SPLINE
SPL {X  -158.456, Y  +360.399, Z    +0.000, E1   -16.490, E3 -394778.901}
SPL {X  -159.553, Y  +370.677, Z    +0.000, E1   -10.576, E3 -394786.661}
SPL {X  -159.960, Y  +379.402, Z    +0.000, E1    -5.303, E3 -394790.682}
SPL {X  -159.990, Y  +385.983, Z    +0.000, E1    -0.882, E3 -394792.754}
SPL {X  -159.990, Y  +390.933, Z    +0.000, E1    +2.877, E3 -394794.202}
SPL {X  -159.990, Y  +396.375, Z    +0.000, E1    +7.538, E3 -394795.977}
SPL {X  -159.990, Y  +405.219, Z    +0.000, E1   +15.296, E3 -394800.294}
SPL {X  -159.990, Y  +427.416, Z    +0.000, E1   +29.294, E3 -394821.349}
SPL {X  -159.990, Y  +450.630, Z    +0.000, E1   +34.875, E3 -394862.921}
SPL {X  -159.990, Y  +456.402, Z    +0.000, E1   +35.061, E3 -394879.197}
SPL {X  -159.990, Y  +460.708, Z    +0.000, E1   +35.045, E3 -394892.255}
SPL {X  -159.990, Y  +464.162, Z    +0.000, E1   +35.038, E3 -394902.711}
SPL {X  -159.990, Y  +467.857, Z    +0.000, E1   +35.053, E3 -394913.868}
SPL {X  -159.990, Y  +471.326, Z    +0.000, E1   +35.038, E3 -394924.363}
SPL {X  -159.990, Y  +474.610, Z    +0.000, E1   +35.053, E3 -394934.262}
SPL {X  -159.990, Y  +478.303, Z    +0.000, E1   +35.049, E3 -394945.435}
SPL {X  -159.990, Y  +482.537, Z    +0.000, E1   +35.066, E3 -394958.226}
SPL {X  -159.990, Y  +487.181, Z    +0.000, E1   +35.054, E3 -394972.309}
SPL {X  -159.990, Y  +492.368, Z    +0.000, E1   +35.076, E3 -394987.981}
SPL {X  -159.990, Y  +497.072, Z    +0.000, E1   +35.040, E3 -395002.277}
SPL {X  -159.990, Y  +500.395, Z    +0.000, E1   +35.033, E3 -395012.340}
SPL {X  -159.990, Y  +505.138, Z    +0.000, E1   +35.092, E3 -395026.576}
SPL {X  -159.990, Y  +510.443, Z    +0.000, E1   +35.051, E3 -395042.695}
SPL {X  -159.990, Y  +514.632, Z    +0.000, E1   +35.050, E3 -395055.365}
SPL {X  -159.990, Y  +518.055, Z    +0.000, E1   +35.037, E3 -395065.734}
SPL {X  -159.990, Y  +521.637, Z    +0.000, E1   +35.056, E3 -395076.544}
SPL {X  -159.990, Y  +526.246, Z    +0.000, E1   +35.065, E3 -395090.447}
SPL {X  -159.990, Y  +531.319, Z    +0.000, E1   +35.072, E3 -395105.803}
SPL {X  -159.990, Y  +537.053, Z    +0.000, E1   +35.083, E3 -395123.136}
SPL {X  -159.990, Y  +542.114, Z    +0.000, E1   +35.053, E3 -395138.482}
SPL {X  -159.990, Y  +545.724, Z    +0.000, E1   +35.043, E3 -395149.407}
SPL {X  -159.990, Y  +549.546, Z    +0.000, E1   +35.061, E3 -395160.931}
SPL {X  -159.990, Y  +554.793, Z    +0.000, E1   +35.100, E3 -395176.695}
SPL {X  -159.990, Y  +560.931, Z    +0.000, E1   +35.098, E3 -395195.256}
SPL {X  -159.990, Y  +566.542, Z    +0.000, E1   +35.080, E3 -395212.264}
SPL {X  -159.990, Y  +571.374, Z    +0.000, E1   +35.070, E3 -395226.888}
SPL {X  -159.990, Y  +575.771, Z    +0.000, E1   +35.064, E3 -395240.193}
SPL {X  -159.990, Y  +579.185, Z    +0.000, E1   +35.047, E3 -395250.541}
SPL {X  -159.990, Y  +581.944, Z    +0.000, E1   +35.051, E3 -395258.879}
SPL {X  -159.990, Y  +585.414, Z    +0.000, E1   +35.059, E3 -395269.362}
SPL {X  -159.990, Y  +590.166, Z    +0.000, E1   +35.084, E3 -395283.690}
SPL {X  -159.990, Y  +595.313, Z    +0.000, E1   +35.073, E3 -395299.269}
SPL {X  -159.990, Y  +600.543, Z    +0.000, E1   +35.091, E3 -395315.051}
SPL {X  -159.990, Y  +605.846, Z    +0.000, E1   +35.077, E3 -395331.102}
SPL {X  -159.990, Y  +609.372, Z    +0.000, E1   +35.047, E3 -395341.800}
SPL {X  -159.990, Y  +613.036, Z    +0.000, E1   +35.082, E3 -395352.835}
SPL {X  -159.990, Y  +617.577, Z    +0.000, E1   +35.061, E3 -395366.596}
SPL {X  -159.990, Y  +621.534, Z    +0.000, E1   +35.068, E3 -395378.531}
SPL {X  -159.990, Y  +625.237, Z    +0.000, E1   +35.062, E3 -395389.733}
SPL {X  -159.990, Y  +629.217, Z    +0.000, E1   +35.065, E3 -395401.790}
SPL {X  -159.990, Y  +632.566, Z    +0.000, E1   +35.044, E3 -395411.953}
SPL {X  -159.990, Y  +635.965, Z    +0.000, E1   +35.065, E3 -395422.196}
SPL {X  -159.990, Y  +640.633, Z    +0.000, E1   +35.080, E3 -395436.285}
SPL {X  -159.990, Y  +646.430, Z    +0.000, E1   +35.102, E3 -395453.786}
SPL {X  -159.990, Y  +651.502, Z    +0.000, E1   +35.058, E3 -395469.196}
SPL {X  -159.990, Y  +654.793, Z    +0.000, E1   +35.049, E3 -395479.159}
SPL {X  -159.990, Y  +657.535, Z    +0.000, E1   +35.049, E3 -395487.456}
SPL {X  -159.990, Y  +661.105, Z    +0.000, E1   +35.059, E3 -395498.236}
SPL {X  -159.990, Y  +665.311, Z    +0.000, E1   +35.064, E3 -395510.951}
SPL {X  -159.990, Y  +670.193, Z    +0.000, E1   +35.076, E3 -395525.698}
SPL {X  -159.948, Y  +675.148, Z    +0.000, E1   +35.069, E3 -395540.690}
SPL {X  -159.752, Y  +680.228, Z    +0.000, E1   +35.050, E3 -395556.238}
SPL {X  -159.371, Y  +685.563, Z    +0.000, E1   +34.989, E3 -395572.749}
SPL {X  -158.886, Y  +690.264, Z    +0.000, E1   +34.888, E3 -395587.500}
SPL {X  -158.362, Y  +694.266, Z    +0.000, E1   +34.794, E3 -395600.174}
SPL {X  -157.614, Y  +698.973, Z    +0.000, E1   +34.690, E3 -395615.174}
SPL {X  -156.640, Y  +704.066, Z    +0.000, E1   +34.516, E3 -395631.600}
SPL {X  -155.835, Y  +707.723, Z    +0.000, E1   +34.344, E3 -395643.542}
SPL {X  -155.080, Y  +710.833, Z    +0.000, E1   +34.231, E3 -395653.692}
SPL {X  -153.755, Y  +715.731, Z    +0.000, E1   +30.246, E3 -395702.958}
ENDSPLINE

SPLINE
SPL {X  -155.537, Y  +708.983, Z    +0.000, E1   +25.008, E3 -395728.784}
SPL {X  -158.838, Y  +690.666, Z    +0.000, E1   +14.584, E3 -395753.497}
SPL {X  -159.750, Y  +680.262, Z    +0.000, E1    +8.563, E3 -395759.637}
SPL {X  -159.973, Y  +673.798, Z    +0.000, E1    +4.600, E3 -395762.101}
SPL {X  -159.990, Y  +668.863, Z    +0.000, E1    +1.298, E3 -395763.541}
SPL {X  -159.990, Y  +663.839, Z    +0.000, E1    -2.454, E3 -395764.802}
SPL {X  -159.990, Y  +657.071, Z    +0.000, E1    -8.297, E3 -395766.994}
SPL {X  -159.990, Y  +646.193, Z    +0.000, E1   -17.980, E3 -395772.721}
SPL {X  -159.990, Y  +621.124, Z    +0.000, E1   -32.598, E3 -395796.208}
SPL {X  -159.990, Y  +597.855, Z    +0.000, E1   -36.862, E3 -395839.127}
SPL {X  -159.990, Y  +592.884, Z    +0.000, E1   -36.865, E3 -395853.198}
SPL {X  -159.990, Y  +587.104, Z    +0.000, E1   -36.878, E3 -395869.555}
SPL {X  -159.990, Y  +581.795, Z    +0.000, E1   -36.847, E3 -395884.654}
SPL {X  -159.990, Y  +576.165, Z    +0.000, E1   -36.887, E3 -395900.533}
SPL {X  -159.990, Y  +570.328, Z    +0.000, E1   -36.855, E3 -395917.106}
SPL {X  -159.990, Y  +566.126, Z    +0.000, E1   -36.841, E3 -395929.012}
SPL {X  -159.990, Y  +562.387, Z    +0.000, E1   -36.853, E3 -395939.545}
SPL {X  -159.990, Y  +557.944, Z    +0.000, E1   -36.859, E3 -395952.139}
SPL {X  -159.990, Y  +553.661, Z    +0.000, E1   -36.844, E3 -395964.303}
SPL {X  -159.990, Y  +549.195, Z    +0.000, E1   -36.856, E3 -395976.938}
SPL {X  -159.990, Y  +543.458, Z    +0.000, E1   -36.882, E3 -395993.136}
SPL {X  -159.990, Y  +538.694, Z    +0.000, E1   -36.835, E3 -396006.720}
SPL {X  -159.990, Y  +534.469, Z    +0.000, E1   -36.855, E3 -396018.666}
SPL {X  -159.990, Y  +530.428, Z    +0.000, E1   -36.821, E3 -396030.199}
SPL {X  -159.990, Y  +525.940, Z    +0.000, E1   -36.859, E3 -396042.846}
SPL {X  -159.990, Y  +520.301, Z    +0.000, E1   -36.855, E3 -396058.822}
SPL {X  -159.990, Y  +516.005, Z    +0.000, E1   -36.824, E3 -396071.048}
SPL {X  -159.990, Y  +512.789, Z    +0.000, E1   -36.824, E3 -396080.156}
SPL {X  -159.990, Y  +508.591, Z    +0.000, E1   -36.846, E3 -396092.019}
SPL {X  -159.990, Y  +503.454, Z    +0.000, E1   -36.847, E3 -396106.574}
SPL {X  -159.990, Y  +498.817, Z    +0.000, E1   -36.830, E3 -396119.757}
SPL {X  -159.990, Y  +498.054, Z    +0.000, E1   -35.692, E3 -396128.871}
ENDSPLINE

SPLINE
SPL {X  -159.990, Y  +505.140, Z    +0.000, E1   -30.523, E3 -396139.898}
ENDSPLINE

SPLINE
SPL {X  -159.990, Y  +497.800, Z    +0.000, E1   -31.845, E3 -396156.854}
SPL {X  -159.990, Y  +492.180, Z    +0.000, E1   -32.851, E3 -396168.990}
SPL {X  -159.990, Y  +486.073, Z    +0.000, E1   -33.960, E3 -396181.625}
SPL {X  -159.990, Y  +477.314, Z    +0.000, E1   -35.342, E3 -396199.803}
SPL {X  -159.990, Y  +471.459, Z    +0.000, E1   -35.779, E3 -396214.343}
SPL {X  -159.990, Y  +467.485, Z    +0.000, E1   -35.768, E3 -396226.072}
SPL {X  -159.990, Y  +462.739, Z    +0.000, E1   -35.799, E3 -396240.000}
SPL {X  -159.990, Y  +457.385, Z    +0.000, E1   -35.788, E3 -396255.784}
SPL {X  -159.990, Y  +452.637, Z    +0.000, E1   -35.783, E3 -396269.776}
SPL {X  -159.990, Y  +446.982, Z    +0.000, E1   -35.815, E3 -396286.377}
SPL {X  -159.990, Y  +442.593, Z    +0.000, E1   -35.759, E3 -396299.386}
SPL {X  -159.990, Y  +439.109, Z    +0.000, E1   -35.781, E3 -396309.603}
SPL {X  -159.990, Y  +435.535, Z    +0.000, E1   -35.764, E3 -396320.154}
SPL {X  -159.990, Y  +431.100, Z    +0.000, E1   -35.807, E3 -396333.139}
SPL {X  -159.990, Y  +426.641, Z    +0.000, E1   -35.769, E3 -396346.326}
SPL {X  -159.990, Y  +422.627, Z    +0.000, E1   -35.788, E3 -396358.123}
SPL {X  -159.990, Y  +417.866, Z    +0.000, E1   -35.788, E3 -396372.137}
SPL {X  -159.990, Y  +413.498, Z    +0.000, E1   -35.779, E3 -396385.019}
SPL {X  -159.990, Y  +408.600, Z    +0.000, E1   -35.802, E3 -396399.406}
SPL {X  -159.990, Y  +403.496, Z    +0.000, E1   -35.787, E3 -396414.461}
SPL {X  -159.990, Y  +398.606, Z    +0.000, E1   -35.794, E3 -396428.848}
SPL {X  -159.990, Y  +394.138, Z    +0.000, E1   -35.778, E3 -396442.032}
SPL {X  -159.990, Y  +388.813, Z    +0.000, E1   -35.819, E3 -396457.644}
SPL {X  -159.990, Y  +383.172, Z    +0.000, E1   -35.789, E3 -396474.298}
SPL {X  -159.936, Y  +378.352, Z    +0.000, E1   -35.782, E3 -396488.537}
SPL {X  -159.790, Y  +374.497, Z    +0.000, E1   -35.735, E3 -396500.081}
SPL {X  -159.547, Y  +370.604, Z    +0.000, E1   -35.724, E3 -396511.766}
SPL {X  -159.134, Y  +365.969, Z    +0.000, E1   -35.644, E3 -396525.852}
SPL {X  -158.606, Y  +361.498, Z    +0.000, E1   -35.550, E3 -396539.616}
SPL {X  -157.918, Y  +356.833, Z    +0.000, E1   -35.439, E3 -396554.069}
SPL {X  -157.185, Y  +352.671, Z    +0.000, E1   -35.292, E3 -396567.129}
SPL {X  -156.302, Y  +348.345, Z    +0.000, E1   -35.165, E3 -396580.750}
SPL {X  -155.054, Y  +343.066, Z    +0.000, E1   -34.964, E3 -396597.565}
SPL {X  -154.305, Y  +340.232, Z    +0.000, E1   -28.975, E3 -396655.125}
ENDSPLINE

SPLINE
SPL {X  -158.456, Y  +360.399, Z    +0.000, E1   -16.490, E3 -396691.945}
SPL {X  -159.553, Y  +370.677, Z    +0.000, E1   -10.576, E3 -396699.705}
SPL {X  -159.960, Y  +379.402, Z    +0.000, E1    -5.303, E3 -396703.725}
SPL {X  -159.990, Y  +387.301, Z    +0.000, E1    -0.001, E3 -396706.186}
SPL {X  -159.990, Y  +392.161, Z    +0.000, E1    +3.946, E3 -396707.598}
SPL {X  -159.990, Y  +396.375, Z    +0.000, E1    +7.538, E3 -396709.020}
SPL {X  -159.990, Y  +404.277, Z    +0.000, E1   +14.543, E3 -396712.683}
SPL {X  -159.990, Y  +423.101, Z    +0.000, E1   +27.351, E3 -396729.122}
SPL {X  -159.990, Y  +430.933, Z    +0.000, E1   +30.672, E3 -396739.093}
SPL {X  -159.990, Y  +451.842, Z    +0.000, E1   +35.050, E3 -396778.464}
SPL {X  -159.990, Y  +456.402, Z    +0.000, E1   +35.061, E3 -396792.240}
SPL {X  -159.990, Y  +460.708, Z    +0.000, E1   +35.045, E3 -396805.298}
SPL {X  -159.990, Y  +464.162, Z    +0.000, E1   +35.038, E3 -396815.754}
SPL {X  -159.990, Y  +467.857, Z    +0.000, E1   +35.053, E3 -396826.911}
SPL {X  -159.990, Y  +471.326, Z    +0.000, E1   +35.038, E3 -396837.406}
SPL {X  -159.990, Y  +474.610, Z    +0.000, E1   +35.053, E3 -396847.306}
SPL {X  -159.990, Y  +478.303, Z    +0.000, E1   +35.049, E3 -396858.478}
SPL {X  -159.990, Y  +482.537, Z    +0.000, E1   +35.066, E3 -396871.269}
SPL {X  -159.990, Y  +487.181, Z    +0.000, E1   +35.054, E3 -396885.352}
SPL {X  -159.990, Y  +490.807, Z    +0.000, E1   +35.036, E3 -396896.354}
SPL {X  -159.990, Y  +493.669, Z    +0.000, E1   +35.034, E3 -396905.033}
SPL {X  -159.990, Y  +497.072, Z    +0.000, E1   +35.040, E3 -396915.320}
SPL {X  -159.990, Y  +501.645, Z    +0.000, E1   +35.067, E3 -396929.103}
SPL {X  -159.990, Y  +507.359, Z    +0.000, E1   +35.080, E3 -396946.360}
SPL {X  -159.990, Y  +512.562, Z    +0.000, E1   +35.055, E3 -396962.142}
SPL {X  -159.990, Y  +517.156, Z    +0.000, E1   +35.059, E3 -396976.024}
SPL {X  -159.990, Y  +521.637, Z    +0.000, E1   +35.056, E3 -396989.587}
SPL {X  -159.990, Y  +525.227, Z    +0.000, E1   +35.041, E3 -397000.448}
SPL {X  -159.990, Y  +529.413, Z    +0.000, E1   +35.072, E3 -397013.077}
SPL {X  -159.990, Y  +534.797, Z    +0.000, E1   +35.069, E3 -397029.377}
SPL {X  -159.990, Y  +538.710, Z    +0.000, E1   +35.033, E3 -397041.274}
SPL {X  -159.990, Y  +542.114, Z    +0.000, E1   +35.053, E3 -397051.526}
SPL {X  -159.990, Y  +546.612, Z    +0.000, E1   +35.065, E3 -397065.097}
SPL {X  -159.990, Y  +551.596, Z    +0.000, E1   +35.079, E3 -397080.132}
SPL {X  -159.990, Y  +557.043, Z    +0.000, E1   +35.087, E3 -397096.554}
SPL {X  -159.990, Y  +562.842, Z    +0.000, E1   +35.098, E3 -397114.087}
SPL {X  -159.990, Y  +568.750, Z    +0.000, E1   +35.087, E3 -397131.972}
SPL {X  -159.990, Y  +574.780, Z    +0.000, E1   +35.101, E3 -397150.183}
SPL {X  -159.990, Y  +580.750, Z    +0.000, E1   +35.087, E3 -397168.259}
SPL {X  -159.990, Y  +585.414, Z    +0.000, E1   +35.059, E3 -397182.405}
SPL {X  -159.990, Y  +588.716, Z    +0.000, E1   +35.047, E3 -397192.408}
SPL {X  -159.990, Y  +592.923, Z    +0.000, E1   +35.084, E3 -397205.072}
SPL {X  -159.990, Y  +598.554, Z    +0.000, E1   +35.088, E3 -397222.091}
SPL {X  -159.990, Y  +603.289, Z    +0.000, E1   +35.068, E3 -397236.419}
SPL {X  -159.990, Y  +607.919, Z    +0.000, E1   +35.079, E3 -397250.408}
SPL {X  -159.990, Y  +613.036, Z    +0.000, E1   +35.082, E3 -397265.878}
SPL {X  -159.990, Y  +617.577, Z    +0.000, E1   +35.061, E3 -397279.640}
SPL {X  -159.990, Y  +621.534, Z    +0.000, E1   +35.068, E3 -397291.574}
SPL {X  -159.990, Y  +626.426, Z    +0.000, E1   +35.093, E3 -397306.333}
SPL {X  -159.990, Y  +631.553, Z    +0.000, E1   +35.068, E3 -397321.891}
SPL {X  -159.990, Y  +636.917, Z    +0.000, E1   +35.095, E3 -397338.070}
SPL {X  -159.990, Y  +641.534, Z    +0.000, E1   +35.053, E3 -397352.098}
SPL {X  -159.990, Y  +646.430, Z    +0.000, E1   +35.102, E3 -397366.829}
SPL {X  -159.990, Y  +651.502, Z    +0.000, E1   +35.058, E3 -397382.239}
SPL {X  -159.990, Y  +654.793, Z    +0.000, E1   +35.049, E3 -397392.203}
SPL {X  -159.990, Y  +657.535, Z    +0.000, E1   +35.049, E3 -397400.499}
SPL {X  -159.990, Y  +661.105, Z    +0.000, E1   +35.059, E3 -397411.279}
SPL {X  -159.990, Y  +665.311, Z    +0.000, E1   +35.064, E3 -397423.994}
SPL {X  -159.990, Y  +670.193, Z    +0.000, E1   +35.076, E3 -397438.741}
SPL {X  -159.948, Y  +675.148, Z    +0.000, E1   +35.069, E3 -397453.733}
SPL {X  -159.752, Y  +680.228, Z    +0.000, E1   +35.050, E3 -397469.281}
SPL {X  -159.371, Y  +685.563, Z    +0.000, E1   +34.989, E3 -397485.793}
SPL {X  -158.886, Y  +690.264, Z    +0.000, E1   +34.888, E3 -397500.544}
SPL {X  -158.362, Y  +694.266, Z    +0.000, E1   +34.794, E3 -397513.217}
SPL {X  -157.614, Y  +698.973, Z    +0.000, E1   +34.690, E3 -397528.218}
SPL {X  -156.640, Y  +704.066, Z    +0.000, E1   +34.516, E3 -397544.643}
SPL {X  -155.835, Y  +707.723, Z    +0.000, E1   +34.344, E3 -397556.585}
SPL {X  -155.080, Y  +710.833, Z    +0.000, E1   +34.231, E3 -397566.735}
SPL {X  -153.755, Y  +715.731, Z    +0.000, E1   +30.246, E3 -397616.001}
ENDSPLINE

SPLINE
SPL {X  -155.537, Y  +708.983, Z    +0.000, E1   +25.008, E3 -397641.828}
SPL {X  -158.838, Y  +690.666, Z    +0.000, E1   +14.584, E3 -397666.540}
SPL {X  -159.750, Y  +680.262, Z    +0.000, E1    +8.563, E3 -397672.681}
SPL {X  -159.973, Y  +673.798, Z    +0.000, E1    +4.600, E3 -397675.145}
SPL {X  -159.990, Y  +668.863, Z    +0.000, E1    +1.298, E3 -397676.584}
SPL {X  -159.990, Y  +663.839, Z    +0.000, E1    -2.454, E3 -397677.845}
SPL {X  -159.990, Y  +657.071, Z    +0.000, E1    -8.297, E3 -397680.038}
SPL {X  -159.990, Y  +646.193, Z    +0.000, E1   -17.980, E3 -397685.764}
SPL {X  -159.990, Y  +621.124, Z    +0.000, E1   -32.598, E3 -397709.251}
SPL {X  -159.990, Y  +599.888, Z    +0.000, E1   -36.828, E3 -397746.491}
SPL {X  -159.990, Y  +595.346, Z    +0.000, E1   -36.880, E3 -397759.257}
SPL {X  -159.990, Y  +589.749, Z    +0.000, E1   -36.860, E3 -397775.130}
SPL {X  -159.990, Y  +585.754, Z    +0.000, E1   -36.838, E3 -397786.485}
SPL {X  -159.990, Y  +581.795, Z    +0.000, E1   -36.847, E3 -397797.697}
SPL {X  -159.990, Y  +576.165, Z    +0.000, E1   -36.887, E3 -397813.577}
SPL {X  -159.990, Y  +570.328, Z    +0.000, E1   -36.855, E3 -397830.150}
SPL {X  -159.990, Y  +566.126, Z    +0.000, E1   -36.841, E3 -397842.056}
SPL {X  -159.990, Y  +562.387, Z    +0.000, E1   -36.853, E3 -397852.589}
SPL {X  -159.990, Y  +557.944, Z    +0.000, E1   -36.859, E3 -397865.182}
SPL {X  -159.990, Y  +552.571, Z    +0.000, E1   -36.873, E3 -397880.386}
SPL {X  -159.990, Y  +548.223, Z    +0.000, E1   -36.832, E3 -397892.777}
SPL {X  -159.990, Y  +543.458, Z    +0.000, E1   -36.882, E3 -397906.180}
SPL {X  -159.990, Y  +538.694, Z    +0.000, E1   -36.835, E3 -397919.764}
SPL {X  -159.990, Y  +534.469, Z    +0.000, E1   -36.855, E3 -397931.709}
SPL {X  -159.990, Y  +530.428, Z    +0.000, E1   -36.821, E3 -397943.243}
SPL {X  -159.990, Y  +525.940, Z    +0.000, E1   -36.859, E3 -397955.889}
SPL {X  -159.990, Y  +520.301, Z    +0.000, E1   -36.855, E3 -397971.865}
SPL {X  -159.990, Y  +516.005, Z    +0.000, E1   -36.824, E3 -397984.092}
SPL {X  -159.990, Y  +512.789, Z    +0.000, E1   -36.824, E3 -397993.200}
SPL {X  -159.990, Y  +508.591, Z    +0.000, E1   -36.846, E3 -398005.062}
SPL {X  -159.990, Y  +503.454, Z    +0.000, E1   -36.847, E3 -398019.617}
SPL {X  -159.990, Y  +498.817, Z    +0.000, E1   -36.830, E3 -398032.800}
SPL {X  -159.990, Y  +498.054, Z    +0.000, E1   -35.692, E3 -398041.914}
ENDSPLINE

SPLINE
SPL {X  -159.990, Y  +506.994, Z    +0.000, E1   -30.162, E3 -398048.576}
ENDSPLINE

SPLINE
SPL {X  -159.990, Y  +502.084, Z    +0.000, E1   -31.057, E3 -398060.227}
SPL {X  -159.990, Y  +494.586, Z    +0.000, E1   -32.444, E3 -398076.831}
SPL {X  -159.990, Y  +487.723, Z    +0.000, E1   -33.658, E3 -398091.283}
SPL {X  -159.990, Y  +481.374, Z    +0.000, E1   -34.706, E3 -398104.487}
SPL {X  -159.990, Y  +475.503, Z    +0.000, E1   -35.597, E3 -398116.540}
SPL {X  -159.990, Y  +471.459, Z    +0.000, E1   -35.779, E3 -398127.386}
SPL {X  -159.990, Y  +467.485, Z    +0.000, E1   -35.768, E3 -398139.116}
SPL {X  -159.990, Y  +462.739, Z    +0.000, E1   -35.799, E3 -398153.044}
SPL {X  -159.990, Y  +458.524, Z    +0.000, E1   -35.761, E3 -398165.517}
SPL {X  -159.990, Y  +453.597, Z    +0.000, E1   -35.819, E3 -398179.937}
SPL {X  -159.990, Y  +448.227, Z    +0.000, E1   -35.776, E3 -398195.815}
SPL {X  -159.990, Y  +443.707, Z    +0.000, E1   -35.784, E3 -398209.111}
SPL {X  -159.990, Y  +439.109, Z    +0.000, E1   -35.781, E3 -398222.647}
SPL {X  -159.990, Y  +434.400, Z    +0.000, E1   -35.789, E3 -398236.502}
SPL {X  -159.990, Y  +430.115, Z    +0.000, E1   -35.777, E3 -398249.118}
SPL {X  -159.990, Y  +425.407, Z    +0.000, E1   -35.800, E3 -398262.958}
SPL {X  -159.990, Y  +421.502, Z    +0.000, E1   -35.761, E3 -398274.519}
SPL {X  -159.990, Y  +417.866, Z    +0.000, E1   -35.788, E3 -398285.180}
SPL {X  -159.990, Y  +413.498, Z    +0.000, E1   -35.779, E3 -398298.062}
SPL {X  -159.990, Y  +408.600, Z    +0.000, E1   -35.802, E3 -398312.450}
SPL {X  -159.990, Y  +403.496, Z    +0.000, E1   -35.787, E3 -398327.505}
SPL {X  -159.990, Y  +398.606, Z    +0.000, E1   -35.794, E3 -398341.892}
SPL {X  -159.990, Y  +394.138, Z    +0.000, E1   -35.778, E3 -398355.075}
SPL {X  -159.990, Y  +390.065, Z    +0.000, E1   -35.780, E3 -398367.065}
SPL {X  -159.990, Y  +385.506, Z    +0.000, E1   -35.789, E3 -398380.471}
SPL {X  -159.976, Y  +380.359, Z    +0.000, E1   -35.797, E3 -398395.620}
SPL {X  -159.831, Y  +375.358, Z    +0.000, E1   -35.763, E3 -398410.510}
SPL {X  -159.613, Y  +371.527, Z    +0.000, E1   -35.709, E3 -398422.065}
SPL {X  -159.203, Y  +366.647, Z    +0.000, E1   -35.680, E3 -398436.798}
SPL {X  -158.715, Y  +362.338, Z    +0.000, E1   -35.547, E3 -398450.103}
SPL {X  -158.237, Y  +358.884, Z    +0.000, E1   -35.480, E3 -398460.760}
SPL {X  -157.724, Y  +355.670, Z    +0.000, E1   -35.371, E3 -398470.794}
SPL {X  -157.185, Y  +352.671, Z    +0.000, E1   -35.292, E3 -398480.173}
SPL {X  -156.582, Y  +349.653, Z    +0.000, E1   -35.175, E3 -398489.706}
SPL {X  -155.743, Y  +345.880, Z    +0.000, E1   -35.068, E3 -398501.633}
SPL {X  -154.759, Y  +341.925, Z    +0.000, E1   -34.868, E3 -398514.339}
SPL {X  -154.305, Y  +340.232, Z    +0.000, E1   -28.975, E3 -398568.168}
ENDSPLINE

SPLINE
SPL {X  -158.456, Y  +360.399, Z    +0.000, E1   -16.490, E3 -398604.988}
SPL {X  -159.553, Y  +370.677, Z    +0.000, E1   -10.576, E3 -398612.748}
SPL {X  -159.960, Y  +379.402, Z    +0.000, E1    -5.303, E3 -398616.769}
SPL {X  -159.990, Y  +385.983, Z    +0.000, E1    -0.882, E3 -398618.841}
SPL {X  -159.990, Y  +390.933, Z    +0.000, E1    +2.877, E3 -398620.289}
SPL {X  -159.990, Y  +396.375, Z    +0.000, E1    +7.538, E3 -398622.064}
SPL {X  -159.990, Y  +404.277, Z    +0.000, E1   +14.543, E3 -398625.727}
SPL {X  -159.990, Y  +423.101, Z    +0.000, E1   +27.351, E3 -398642.165}
SPL {X  -159.990, Y  +430.933, Z    +0.000, E1   +30.672, E3 -398652.136}
SPL {X  -159.990, Y  +451.842, Z    +0.000, E1   +35.050, E3 -398691.508}
SPL {X  -159.990, Y  +456.402, Z    +0.000, E1   +35.061, E3 -398705.284}
SPL {X  -159.990, Y  +460.708, Z    +0.000, E1   +35.045, E3 -398718.342}
SPL {X  -159.990, Y  +464.162, Z    +0.000, E1   +35.038, E3 -398728.798}
SPL {X  -159.990, Y  +467.857, Z    +0.000, E1   +35.053, E3 -398739.955}
SPL {X  -159.990, Y  +471.326, Z    +0.000, E1   +35.038, E3 -398750.450}
SPL {X  -159.990, Y  +474.610, Z    +0.000, E1   +35.053, E3 -398760.349}
SPL {X  -159.990, Y  +478.303, Z    +0.000, E1   +35.049, E3 -398771.522}
SPL {X  -159.990, Y  +482.537, Z    +0.000, E1   +35.066, E3 -398784.313}
SPL {X  -159.990, Y  +487.181, Z    +0.000, E1   +35.054, E3 -398798.396}
SPL {X  -159.990, Y  +492.368, Z    +0.000, E1   +35.076, E3 -398814.068}
SPL {X  -159.990, Y  +497.072, Z    +0.000, E1   +35.040, E3 -398828.364}
SPL {X  -159.990, Y  +500.395, Z    +0.000, E1   +35.033, E3 -398838.426}
SPL {X  -159.990, Y  +505.138, Z    +0.000, E1   +35.092, E3 -398852.663}
SPL {X  -159.990, Y  +510.443, Z    +0.000, E1   +35.051, E3 -398868.782}
SPL {X  -159.990, Y  +514.632, Z    +0.000, E1   +35.050, E3 -398881.452}
SPL {X  -159.990, Y  +518.055, Z    +0.000, E1   +35.037, E3 -398891.821}
SPL {X  -159.990, Y  +521.637, Z    +0.000, E1   +35.056, E3 -398902.631}
SPL {X  -159.990, Y  +526.246, Z    +0.000, E1   +35.065, E3 -398916.534}
SPL {X  -159.990, Y  +530.289, Z    +0.000, E1   +35.044, E3 -398928.820}
SPL {X  -159.990, Y  +534.797, Z    +0.000, E1   +35.069, E3 -398942.420}
SPL {X  -159.990, Y  +538.710, Z    +0.000, E1   +35.033, E3 -398954.317}
SPL {X  -159.990, Y  +542.114, Z    +0.000, E1   +35.053, E3 -398964.569}
SPL {X  -159.990, Y  +545.724, Z    +0.000, E1   +35.043, E3 -398975.494}
SPL {X  -159.990, Y  +549.546, Z    +0.000, E1   +35.061, E3 -398987.018}
SPL {X  -159.990, Y  +554.793, Z    +0.000, E1   +35.100, E3 -399002.782}
SPL {X  -159.990, Y  +560.931, Z    +0.000, E1   +35.098, E3 -399021.343}
SPL {X  -159.990, Y  +566.542, Z    +0.000, E1   +35.080, E3 -399038.351}
SPL {X  -159.990, Y  +570.261, Z    +0.000, E1   +35.046, E3 -399049.647}
SPL {X  -159.990, Y  +574.780, Z    +0.000, E1   +35.101, E3 -399063.227}
SPL {X  -159.990, Y  +580.750, Z    +0.000, E1   +35.087, E3 -399081.302}
SPL {X  -159.990, Y  +585.414, Z    +0.000, E1   +35.059, E3 -399095.449}
SPL {X  -159.990, Y  +588.716, Z    +0.000, E1   +35.047, E3 -399105.451}
SPL {X  -159.990, Y  +591.475, Z    +0.000, E1   +35.047, E3 -399113.792}
SPL {X  -159.990, Y  +595.313, Z    +0.000, E1   +35.073, E3 -399125.356}
SPL {X  -159.990, Y  +599.479, Z    +0.000, E1   +35.059, E3 -399137.973}
SPL {X  -159.990, Y  +603.289, Z    +0.000, E1   +35.068, E3 -399149.462}
SPL {X  -159.990, Y  +607.919, Z    +0.000, E1   +35.079, E3 -399163.451}
SPL {X  -159.990, Y  +612.068, Z    +0.000, E1   +35.057, E3 -399176.031}
SPL {X  -159.990, Y  +616.690, Z    +0.000, E1   +35.089, E3 -399189.958}
SPL {X  -159.990, Y  +621.534, Z    +0.000, E1   +35.068, E3 -399204.618}
SPL {X  -159.990, Y  +625.237, Z    +0.000, E1   +35.062, E3 -399215.820}
SPL {X  -159.990, Y  +629.217, Z    +0.000, E1   +35.065, E3 -399227.877}
SPL {X  -159.990, Y  +632.566, Z    +0.000, E1   +35.044, E3 -399238.040}
SPL {X  -159.990, Y  +635.965, Z    +0.000, E1   +35.065, E3 -399248.283}
SPL {X  -159.990, Y  +640.633, Z    +0.000, E1   +35.080, E3 -399262.372}
SPL {X  -159.990, Y  +646.430, Z    +0.000, E1   +35.102, E3 -399279.873}
SPL {X  -159.990, Y  +651.502, Z    +0.000, E1   +35.058, E3 -399295.283}
SPL {X  -159.990, Y  +654.793, Z    +0.000, E1   +35.049, E3 -399305.246}
SPL {X  -159.990, Y  +657.535, Z    +0.000, E1   +35.049, E3 -399313.543}
SPL {X  -159.990, Y  +661.105, Z    +0.000, E1   +35.059, E3 -399324.323}
SPL {X  -159.990, Y  +665.311, Z    +0.000, E1   +35.064, E3 -399337.038}
SPL {X  -159.990, Y  +670.193, Z    +0.000, E1   +35.076, E3 -399351.785}
SPL {X  -159.948, Y  +675.148, Z    +0.000, E1   +35.069, E3 -399366.777}
SPL {X  -159.752, Y  +680.228, Z    +0.000, E1   +35.050, E3 -399382.324}
SPL {X  -159.371, Y  +685.563, Z    +0.000, E1   +34.989, E3 -399398.836}
SPL {X  -158.886, Y  +690.264, Z    +0.000, E1   +34.888, E3 -399413.587}
SPL {X  -158.362, Y  +694.266, Z    +0.000, E1   +34.794, E3 -399426.261}
SPL {X  -157.614, Y  +698.973, Z    +0.000, E1   +34.690, E3 -399441.261}
SPL {X  -156.640, Y  +704.066, Z    +0.000, E1   +34.516, E3 -399457.687}
SPL {X  -155.835, Y  +707.723, Z    +0.000, E1   +34.344, E3 -399469.629}
SPL {X  -155.080, Y  +710.833, Z    +0.000, E1   +34.231, E3 -399479.779}
SPL {X  -153.755, Y  +715.731, Z    +0.000, E1   +30.246, E3 -399529.045}
ENDSPLINE

SPLINE
SPL {X  -155.537, Y  +708.983, Z    +0.000, E1   +25.008, E3 -399554.871}
SPL {X  -158.838, Y  +690.666, Z    +0.000, E1   +14.584, E3 -399579.584}
SPL {X  -159.750, Y  +680.262, Z    +0.000, E1    +8.563, E3 -399585.724}
SPL {X  -159.973, Y  +673.798, Z    +0.000, E1    +4.600, E3 -399588.188}
SPL {X  -159.990, Y  +668.863, Z    +0.000, E1    +1.298, E3 -399589.628}
SPL {X  -159.990, Y  +663.839, Z    +0.000, E1    -2.454, E3 -399590.889}
SPL {X  -159.990, Y  +657.071, Z    +0.000, E1    -8.297, E3 -399593.081}
SPL {X  -159.990, Y  +646.193, Z    +0.000, E1   -17.980, E3 -399598.808}
SPL {X  -159.990, Y  +621.124, Z    +0.000, E1   -32.598, E3 -399622.295}
SPL {X  -159.990, Y  +597.855, Z    +0.000, E1   -36.862, E3 -399665.214}
SPL {X  -159.990, Y  +592.884, Z    +0.000, E1   -36.865, E3 -399679.285}
SPL {X  -159.990, Y  +587.104, Z    +0.000, E1   -36.878, E3 -399695.642}
SPL {X  -159.990, Y  +581.795, Z    +0.000, E1   -36.847, E3 -399710.740}
SPL {X  -159.990, Y  +577.286, Z    +0.000, E1   -36.853, E3 -399723.497}
SPL {X  -159.990, Y  +572.409, Z    +0.000, E1   -36.854, E3 -399737.310}
SPL {X  -159.990, Y  +567.110, Z    +0.000, E1   -36.868, E3 -399752.271}
SPL {X  -159.990, Y  +562.387, Z    +0.000, E1   -36.853, E3 -399765.632}
SPL {X  -159.990, Y  +557.944, Z    +0.000, E1   -36.859, E3 -399778.226}
SPL {X  -159.990, Y  +552.571, Z    +0.000, E1   -36.873, E3 -399793.430}
SPL {X  -159.990, Y  +546.127, Z    +0.000, E1   -36.890, E3 -399811.656}
SPL {X  -159.990, Y  +541.662, Z    +0.000, E1   -36.835, E3 -399824.373}
SPL {X  -159.990, Y  +537.639, Z    +0.000, E1   -36.860, E3 -399835.761}
SPL {X  -159.990, Y  +531.894, Z    +0.000, E1   -36.865, E3 -399852.050}
SPL {X  -159.990, Y  +527.151, Z    +0.000, E1   -36.828, E3 -399865.549}
SPL {X  -159.990, Y  +522.641, Z    +0.000, E1   -36.854, E3 -399878.282}
SPL {X  -159.990, Y  +517.225, Z    +0.000, E1   -36.859, E3 -399893.616}
SPL {X  -159.990, Y  +512.789, Z    +0.000, E1   -36.824, E3 -399906.243}
SPL {X  -159.990, Y  +508.591, Z    +0.000, E1   -36.846, E3 -399918.106}
SPL {X  -159.990, Y  +504.505, Z    +0.000, E1   -36.824, E3 -399929.710}
SPL {X  -159.990, Y  +499.829, Z    +0.000, E1   -36.864, E3 -399942.919}
SPL {X  -159.990, Y  +498.054, Z    +0.000, E1   -35.692, E3 -399954.958}
ENDSPLINE

SPLINE
SPL {X  -159.990, Y  +505.140, Z    +0.000, E1   -30.523, E3 -399965.985}
ENDSPLINE

SPLINE
SPL {X  -159.990, Y  +497.800, Z    +0.000, E1   -31.845, E3 -399982.941}
SPL {X  -159.990, Y  +492.180, Z    +0.000, E1   -32.851, E3 -399995.076}
SPL {X  -159.990, Y  +486.073, Z    +0.000, E1   -33.960, E3 -400007.712}
SPL {X  -159.990, Y  +477.314, Z    +0.000, E1   -35.342, E3 -400025.890}
SPL {X  -159.990, Y  +471.459, Z    +0.000, E1   -35.779, E3 -400040.430}
SPL {X  -159.990, Y  +467.485, Z    +0.000, E1   -35.768, E3 -400052.159}
SPL {X  -159.990, Y  +462.739, Z    +0.000, E1   -35.799, E3 -400066.087}
SPL {X  -159.990, Y  +458.524, Z    +0.000, E1   -35.761, E3 -400078.561}
SPL {X  -159.990, Y  +453.597, Z    +0.000, E1   -35.819, E3 -400092.981}
SPL {X  -159.990, Y  +448.227, Z    +0.000, E1   -35.776, E3 -400108.859}
SPL {X  -159.990, Y  +443.707, Z    +0.000, E1   -35.784, E3 -400122.154}
SPL {X  -159.990, Y  +439.109, Z    +0.000, E1   -35.781, E3 -400135.690}
SPL {X  -159.990, Y  +435.535, Z    +0.000, E1   -35.764, E3 -400146.241}
SPL {X  -159.990, Y  +431.100, Z    +0.000, E1   -35.807, E3 -400159.226}
SPL {X  -159.990, Y  +426.641, Z    +0.000, E1   -35.769, E3 -400172.413}
SPL {X  -159.990, Y  +422.627, Z    +0.000, E1   -35.788, E3 -400184.210}
SPL {X  -159.990, Y  +417.866, Z    +0.000, E1   -35.788, E3 -400198.224}
SPL {X  -159.990, Y  +413.498, Z    +0.000, E1   -35.779, E3 -400211.105}
SPL {X  -159.990, Y  +408.600, Z    +0.000, E1   -35.802, E3 -400225.493}
SPL {X  -159.990, Y  +403.496, Z    +0.000, E1   -35.787, E3 -400240.548}
SPL {X  -159.990, Y  +399.680, Z    +0.000, E1   -35.767, E3 -400251.821}
SPL {X  -159.990, Y  +395.017, Z    +0.000, E1   -35.806, E3 -400265.488}
SPL {X  -159.990, Y  +390.065, Z    +0.000, E1   -35.780, E3 -400280.109}
SPL {X  -159.990, Y  +385.506, Z    +0.000, E1   -35.789, E3 -400293.514}
SPL {X  -159.989, Y  +381.970, Z    +0.000, E1   -35.761, E3 -400303.969}
SPL {X  -159.936, Y  +378.352, Z    +0.000, E1   -35.782, E3 -400314.624}
SPL {X  -159.790, Y  +374.497, Z    +0.000, E1   -35.735, E3 -400326.168}
SPL {X  -159.547, Y  +370.604, Z    +0.000, E1   -35.724, E3 -400337.853}
SPL {X  -159.134, Y  +365.969, Z    +0.000, E1   -35.644, E3 -400351.939}
SPL {X  -158.715, Y  +362.338, Z    +0.000, E1   -35.547, E3 -400363.147}
SPL {X  -158.237, Y  +358.884, Z    +0.000, E1   -35.480, E3 -400373.803}
SPL {X  -157.724, Y  +355.670, Z    +0.000, E1   -35.371, E3 -400383.838}
SPL {X  -157.185, Y  +352.671, Z    +0.000, E1   -35.292, E3 -400393.216}
SPL {X  -156.302, Y  +348.345, Z    +0.000, E1   -35.165, E3 -400406.837}
SPL {X  -155.054, Y  +343.066, Z    +0.000, E1   -34.964, E3 -400423.652}
SPL {X  -154.305, Y  +340.232, Z    +0.000, E1   -28.975, E3 -400481.212}
ENDSPLINE

SPLINE
SPL {X  -158.456, Y  +360.399, Z    +0.000, E1   -16.490, E3 -400518.032}
SPL {X  -159.553, Y  +370.677, Z    +0.000, E1   -10.576, E3 -400525.792}
SPL {X  -159.960, Y  +379.402, Z    +0.000, E1    -5.303, E3 -400529.812}
SPL {X  -159.990, Y  +387.301, Z    +0.000, E1    -0.001, E3 -400532.273}
SPL {X  -159.990, Y  +392.161, Z    +0.000, E1    +3.946, E3 -400533.685}
SPL {X  -159.990, Y  +396.375, Z    +0.000, E1    +7.538, E3 -400535.107}
SPL {X  -159.990, Y  +404.277, Z    +0.000, E1   +14.543, E3 -400538.770}
SPL {X  -159.990, Y  +423.101, Z    +0.000, E1   +27.351, E3 -400555.209}
SPL {X  -159.990, Y  +430.933, Z    +0.000, E1   +30.672, E3 -400565.180}
SPL {X  -159.990, Y  +451.842, Z    +0.000, E1   +35.050, E3 -400604.551}
SPL {X  -159.990, Y  +456.402, Z    +0.000, E1   +35.061, E3 -400618.327}
SPL {X  -159.990, Y  +460.708, Z    +0.000, E1   +35.045, E3 -400631.385}
SPL {X  -159.990, Y  +464.162, Z    +0.000, E1   +35.038, E3 -400641.841}
SPL {X  -159.990, Y  +467.857, Z    +0.000, E1   +35.053, E3 -400652.998}
SPL {X  -159.990, Y  +471.326, Z    +0.000, E1   +35.038, E3 -400663.493}
SPL {X  -159.990, Y  +474.610, Z    +0.000, E1   +35.053, E3 -400673.393}
SPL {X  -159.990, Y  +478.303, Z    +0.000, E1   +35.049, E3 -400684.565}
SPL {X  -159.990, Y  +482.537, Z    +0.000, E1   +35.066, E3 -400697.356}
SPL {X  -159.990, Y  +487.181, Z    +0.000, E1   +35.054, E3 -400711.439}
SPL {X  -159.990, Y  +492.368, Z    +0.000, E1   +35.076, E3 -400727.111}
SPL {X  -159.990, Y  +497.072, Z    +0.000, E1   +35.040, E3 -400741.407}
SPL {X  -159.990, Y  +501.645, Z    +0.000, E1   +35.067, E3 -400755.190}
SPL {X  -159.990, Y  +506.307, Z    +0.000, E1   +35.049, E3 -400769.312}
SPL {X  -159.990, Y  +511.643, Z    +0.000, E1   +35.091, E3 -400785.392}
SPL {X  -159.990, Y  +517.156, Z    +0.000, E1   +35.059, E3 -400802.111}
SPL {X  -159.990, Y  +521.637, Z    +0.000, E1   +35.056, E3 -400815.674}
SPL {X  -159.990, Y  +526.246, Z    +0.000, E1   +35.065, E3 -400829.577}
SPL {X  -159.990, Y  +531.319, Z    +0.000, E1   +35.072, E3 -400844.934}
SPL {X  -159.990, Y  +537.053, Z    +0.000, E1   +35.083, E3 -400862.266}
SPL {X  -159.990, Y  +542.114, Z    +0.000, E1   +35.053, E3 -400877.613}
SPL {X  -159.990, Y  +546.612, Z    +0.000, E1   +35.065, E3 -400891.184}
SPL {X  -159.990, Y  +551.596, Z    +0.000, E1   +35.079, E3 -400906.219}
SPL {X  -159.990, Y  +557.043, Z    +0.000, E1   +35.087, E3 -400922.641}
SPL {X  -159.990, Y  +561.808, Z    +0.000, E1   +35.066, E3 -400937.094}
SPL {X  -159.990, Y  +566.542, Z    +0.000, E1   +35.080, E3 -400951.394}
SPL {X  -159.990, Y  +571.374, Z    +0.000, E1   +35.070, E3 -400966.018}
SPL {X  -159.990, Y  +575.771, Z    +0.000, E1   +35.064, E3 -400979.323}
SPL {X  -159.990, Y  +580.750, Z    +0.000, E1   +35.087, E3 -400994.346}
SPL {X  -159.990, Y  +585.414, Z    +0.000, E1   +35.059, E3 -401008.492}
SPL {X  -159.990, Y  +590.166, Z    +0.000, E1   +35.084, E3 -401022.821}
SPL {X  -159.990, Y  +595.313, Z    +0.000, E1   +35.073, E3 -401038.399}
SPL {X  -159.990, Y  +600.543, Z    +0.000, E1   +35.091, E3 -401054.182}
SPL {X  -159.990, Y  +605.846, Z    +0.000, E1   +35.077, E3 -401070.233}
SPL {X  -159.990, Y  +611.113, Z    +0.000, E1   +35.087, E3 -401086.138}
SPL {X  -159.990, Y  +616.690, Z    +0.000, E1   +35.089, E3 -401103.002}
SPL {X  -159.990, Y  +621.534, Z    +0.000, E1   +35.068, E3 -401117.661}
SPL {X  -159.990, Y  +626.426, Z    +0.000, E1   +35.093, E3 -401132.420}
SPL {X  -159.990, Y  +631.553, Z    +0.000, E1   +35.068, E3 -401147.978}
SPL {X  -159.990, Y  +635.965, Z    +0.000, E1   +35.065, E3 -401161.327}
SPL {X  -159.990, Y  +640.633, Z    +0.000, E1   +35.080, E3 -401175.415}
SPL {X  -159.990, Y  +646.430, Z    +0.000, E1   +35.102, E3 -401192.916}
SPL {X  -159.990, Y  +651.502, Z    +0.000, E1   +35.058, E3 -401208.326}
SPL {X  -159.990, Y  +656.270, Z    +0.000, E1   +35.087, E3 -401222.703}
SPL {X  -159.990, Y  +661.105, Z    +0.000, E1   +35.059, E3 -401237.366}
SPL {X  -159.990, Y  +665.311, Z    +0.000, E1   +35.064, E3 -401250.081}
SPL {X  -159.990, Y  +670.193, Z    +0.000, E1   +35.076, E3 -401264.828}
SPL {X  -159.948, Y  +675.148, Z    +0.000, E1   +35.069, E3 -401279.820}
SPL {X  -159.752, Y  +680.228, Z    +0.000, E1   +35.050, E3 -401295.368}
SPL {X  -159.371, Y  +685.563, Z    +0.000, E1   +34.989, E3 -401311.880}
SPL {X  -158.886, Y  +690.264, Z    +0.000, E1   +34.888, E3 -401326.631}
SPL {X  -158.362, Y  +694.266, Z    +0.000, E1   +34.794, E3 -401339.304}
SPL {X  -157.614, Y  +698.973, Z    +0.000, E1   +34.690, E3 -401354.305}
SPL {X  -156.901, Y  +702.787, Z    +0.000, E1   +34.523, E3 -401366.648}
SPL {X  -156.097, Y  +706.580, Z    +0.000, E1   +34.427, E3 -401378.888}
SPL {X  -155.080, Y  +710.833, Z    +0.000, E1   +34.231, E3 -401392.822}
SPL {X  -153.755, Y  +715.731, Z    +0.000, E1   +30.246, E3 -401442.088}
ENDSPLINE

SPLINE
SPL {X  -155.537, Y  +708.983, Z    +0.000, E1   +25.008, E3 -401467.915}
SPL {X  -158.838, Y  +690.666, Z    +0.000, E1   +14.584, E3 -401492.627}
SPL {X  -159.750, Y  +680.262, Z    +0.000, E1    +8.563, E3 -401498.768}
SPL {X  -159.973, Y  +673.798, Z    +0.000, E1    +4.600, E3 -401501.232}
SPL {X  -159.990, Y  +667.448, Z    +0.000, E1    +0.356, E3 -401503.011}
SPL {X  -159.990, Y  +662.686, Z    +0.000, E1    -3.472, E3 -401504.246}
SPL {X  -159.990, Y  +657.071, Z    +0.000, E1    -8.297, E3 -401506.125}
SPL {X  -159.990, Y  +646.193, Z    +0.000, E1   -17.980, E3 -401511.851}
SPL {X  -159.990, Y  +621.124, Z    +0.000, E1   -32.598, E3 -401535.338}
SPL {X  -159.990, Y  +597.855, Z    +0.000, E1   -36.862, E3 -401578.257}
SPL {X  -159.990, Y  +592.884, Z    +0.000, E1   -36.865, E3 -401592.328}
SPL {X  -159.990, Y  +587.104, Z    +0.000, E1   -36.878, E3 -401608.685}
SPL {X  -159.990, Y  +581.795, Z    +0.000, E1   -36.847, E3 -401623.784}
SPL {X  -159.990, Y  +576.165, Z    +0.000, E1   -36.887, E3 -401639.664}
SPL {X  -159.990, Y  +570.328, Z    +0.000, E1   -36.855, E3 -401656.237}
SPL {X  -159.990, Y  +566.126, Z    +0.000, E1   -36.841, E3 -401668.143}
SPL {X  -159.990, Y  +562.387, Z    +0.000, E1   -36.853, E3 -401678.676}
SPL {X  -159.990, Y  +557.944, Z    +0.000, E1   -36.859, E3 -401691.269}
SPL {X  -159.990, Y  +553.661, Z    +0.000, E1   -36.844, E3 -401703.433}
SPL {X  -159.990, Y  +549.195, Z    +0.000, E1   -36.856, E3 -401716.068}
SPL {X  -159.990, Y  +544.733, Z    +0.000, E1   -36.845, E3 -401728.714}
SPL {X  -159.990, Y  +539.889, Z    +0.000, E1   -36.872, E3 -401742.399}
SPL {X  -159.990, Y  +534.469, Z    +0.000, E1   -36.855, E3 -401757.796}
SPL {X  -159.990, Y  +530.428, Z    +0.000, E1   -36.821, E3 -401769.330}
SPL {X  -159.990, Y  +525.940, Z    +0.000, E1   -36.859, E3 -401781.976}
SPL {X  -159.990, Y  +520.301, Z    +0.000, E1   -36.855, E3 -401797.952}
SPL {X  -159.990, Y  +514.308, Z    +0.000, E1   -36.869, E3 -401814.915}
SPL {X  -159.990, Y  +508.591, Z    +0.000, E1   -36.846, E3 -401831.149}
SPL {X  -159.990, Y  +503.454, Z    +0.000, E1   -36.847, E3 -401845.704}
SPL {X  -159.990, Y  +498.817, Z    +0.000, E1   -36.830, E3 -401858.887}
SPL {X  -159.990, Y  +498.054, Z    +0.000, E1   -35.692, E3 -401868.001}
ENDSPLINE

SPLINE
SPL {X  -159.990, Y  +506.994, Z    +0.000, E1   -30.162, E3 -401874.663}
ENDSPLINE

SPLINE
SPL {X  -159.990, Y  +502.084, Z    +0.000, E1   -31.057, E3 -401886.314}
SPL {X  -159.990, Y  +494.586, Z    +0.000, E1   -32.444, E3 -401902.918}
SPL {X  -159.990, Y  +486.073, Z    +0.000, E1   -33.960, E3 -401920.755}
SPL {X  -159.990, Y  +477.314, Z    +0.000, E1   -35.342, E3 -401938.934}
SPL {X  -159.990, Y  +471.459, Z    +0.000, E1   -35.779, E3 -401953.473}
SPL {X  -159.990, Y  +467.485, Z    +0.000, E1   -35.768, E3 -401965.203}
SPL {X  -159.990, Y  +462.739, Z    +0.000, E1   -35.799, E3 -401979.131}
SPL {X  -159.990, Y  +457.385, Z    +0.000, E1   -35.788, E3 -401994.914}
SPL {X  -159.990, Y  +452.637, Z    +0.000, E1   -35.783, E3 -402008.906}
SPL {X  -159.990, Y  +446.982, Z    +0.000, E1   -35.815, E3 -402025.507}
SPL {X  -159.990, Y  +442.593, Z    +0.000, E1   -35.759, E3 -402038.516}
SPL {X  -159.990, Y  +439.109, Z    +0.000, E1   -35.781, E3 -402048.734}
SPL {X  -159.990, Y  +434.400, Z    +0.000, E1   -35.789, E3 -402062.589}
SPL {X  -159.990, Y  +430.115, Z    +0.000, E1   -35.777, E3 -402075.205}
SPL {X  -159.990, Y  +426.641, Z    +0.000, E1   -35.769, E3 -402085.456}
SPL {X  -159.990, Y  +422.627, Z    +0.000, E1   -35.788, E3 -402097.254}
SPL {X  -159.990, Y  +419.027, Z    +0.000, E1   -35.762, E3 -402107.894}
SPL {X  -159.990, Y  +414.514, Z    +0.000, E1   -35.815, E3 -402121.098}
SPL {X  -159.990, Y  +408.600, Z    +0.000, E1   -35.802, E3 -402138.537}
SPL {X  -159.990, Y  +403.496, Z    +0.000, E1   -35.787, E3 -402153.592}
SPL {X  -159.990, Y  +398.606, Z    +0.000, E1   -35.794, E3 -402167.979}
SPL {X  -159.990, Y  +394.138, Z    +0.000, E1   -35.778, E3 -402181.162}
SPL {X  -159.990, Y  +390.065, Z    +0.000, E1   -35.780, E3 -402193.152}
SPL {X  -159.990, Y  +386.815, Z    +0.000, E1   -35.761, E3 -402202.745}
SPL {X  -159.990, Y  +383.172, Z    +0.000, E1   -35.789, E3 -402213.428}
SPL {X  -159.936, Y  +378.352, Z    +0.000, E1   -35.782, E3 -402227.667}
SPL {X  -159.693, Y  +372.749, Z    +0.000, E1   -35.767, E3 -402244.400}
SPL {X  -159.203, Y  +366.647, Z    +0.000, E1   -35.680, E3 -402262.885}
SPL {X  -158.715, Y  +362.338, Z    +0.000, E1   -35.547, E3 -402276.190}
SPL {X  -158.237, Y  +358.884, Z    +0.000, E1   -35.480, E3 -402286.847}
SPL {X  -157.724, Y  +355.670, Z    +0.000, E1   -35.371, E3 -402296.881}
SPL {X  -157.185, Y  +352.671, Z    +0.000, E1   -35.292, E3 -402306.260}
SPL {X  -156.302, Y  +348.345, Z    +0.000, E1   -35.165, E3 -402319.881}
SPL {X  -155.054, Y  +343.066, Z    +0.000, E1   -34.964, E3 -402336.696}
SPL {X  -154.305, Y  +340.232, Z    +0.000, E1   -28.975, E3 -402394.255}
ENDSPLINE

SPLINE
SPL {X  -158.456, Y  +360.399, Z    +0.000, E1   -16.490, E3 -402431.075}
SPL {X  -159.553, Y  +370.677, Z    +0.000, E1   -10.576, E3 -402438.835}
SPL {X  -159.960, Y  +379.402, Z    +0.000, E1    -5.303, E3 -402442.856}
SPL {X  -159.990, Y  +385.983, Z    +0.000, E1    -0.882, E3 -402444.928}
SPL {X  -159.990, Y  +390.933, Z    +0.000, E1    +2.877, E3 -402446.376}
SPL {X  -159.990, Y  +396.375, Z    +0.000, E1    +7.538, E3 -402448.151}
SPL {X  -159.990, Y  +404.277, Z    +0.000, E1   +14.543, E3 -402451.814}
SPL {X  -159.990, Y  +423.101, Z    +0.000, E1   +27.351, E3 -402468.252}
SPL {X  -159.990, Y  +430.396, Z    +0.000, E1   +30.473, E3 -402477.506}
SPL {X  -159.990, Y  +450.630, Z    +0.000, E1   +34.875, E3 -402515.095}
SPL {X  -159.990, Y  +456.402, Z    +0.000, E1   +35.061, E3 -402531.371}
SPL {X  -159.990, Y  +460.708, Z    +0.000, E1   +35.045, E3 -402544.428}
SPL {X  -159.990, Y  +465.240, Z    +0.000, E1   +35.066, E3 -402558.104}
SPL {X  -159.990, Y  +470.278, Z    +0.000, E1   +35.063, E3 -402573.338}
SPL {X  -159.990, Y  +474.610, Z    +0.000, E1   +35.053, E3 -402586.436}
SPL {X  -159.990, Y  +478.303, Z    +0.000, E1   +35.049, E3 -402597.609}
SPL {X  -159.990, Y  +482.537, Z    +0.000, E1   +35.066, E3 -402610.400}
SPL {X  -159.990, Y  +487.181, Z    +0.000, E1   +35.054, E3 -402624.483}
SPL {X  -159.990, Y  +492.368, Z    +0.000, E1   +35.076, E3 -402640.155}
SPL {X  -159.990, Y  +497.072, Z    +0.000, E1   +35.040, E3 -402654.451}
SPL {X  -159.990, Y  +501.645, Z    +0.000, E1   +35.067, E3 -402668.234}
SPL {X  -159.990, Y  +507.359, Z    +0.000, E1   +35.080, E3 -402685.491}
SPL {X  -159.990, Y  +512.562, Z    +0.000, E1   +35.055, E3 -402701.273}
SPL {X  -159.990, Y  +517.156, Z    +0.000, E1   +35.059, E3 -402715.154}
SPL {X  -159.990, Y  +521.637, Z    +0.000, E1   +35.056, E3 -402728.718}
SPL {X  -159.990, Y  +526.246, Z    +0.000, E1   +35.065, E3 -402742.621}
SPL {X  -159.990, Y  +531.319, Z    +0.000, E1   +35.072, E3 -402757.977}
SPL {X  -159.990, Y  +537.053, Z    +0.000, E1   +35.083, E3 -402775.310}
SPL {X  -159.990, Y  +542.114, Z    +0.000, E1   +35.053, E3 -402790.656}
SPL {X  -159.990, Y  +546.612, Z    +0.000, E1   +35.065, E3 -402804.228}
SPL {X  -159.990, Y  +551.596, Z    +0.000, E1   +35.079, E3 -402819.263}
SPL {X  -159.990, Y  +557.043, Z    +0.000, E1   +35.087, E3 -402835.685}
SPL {X  -159.990, Y  +561.808, Z    +0.000, E1   +35.066, E3 -402850.138}
SPL {X  -159.990, Y  +566.542, Z    +0.000, E1   +35.080, E3 -402864.438}
SPL {X  -159.990, Y  +571.374, Z    +0.000, E1   +35.070, E3 -402879.062}
SPL {X  -159.990, Y  +575.771, Z    +0.000, E1   +35.064, E3 -402892.367}
SPL {X  -159.990, Y  +580.750, Z    +0.000, E1   +35.087, E3 -402907.389}
SPL {X  -159.990, Y  +585.414, Z    +0.000, E1   +35.059, E3 -402921.536}
SPL {X  -159.990, Y  +590.166, Z    +0.000, E1   +35.084, E3 -402935.864}
SPL {X  -159.990, Y  +595.313, Z    +0.000, E1   +35.073, E3 -402951.443}
SPL {X  -159.990, Y  +600.543, Z    +0.000, E1   +35.091, E3 -402967.225}
SPL {X  -159.990, Y  +605.846, Z    +0.000, E1   +35.077, E3 -402983.276}
SPL {X  -159.990, Y  +611.113, Z    +0.000, E1   +35.087, E3 -402999.182}
SPL {X  -159.990, Y  +616.690, Z    +0.000, E1   +35.089, E3 -403016.045}
SPL {X  -159.990, Y  +621.534, Z    +0.000, E1   +35.068, E3 -403030.705}
SPL {X  -159.990, Y  +626.426, Z    +0.000, E1   +35.093, E3 -403045.464}
SPL {X  -159.990, Y  +631.553, Z    +0.000, E1   +35.068, E3 -403061.022}
SPL {X  -159.990, Y  +635.965, Z    +0.000, E1   +35.065, E3 -403074.370}
SPL {X  -159.990, Y  +640.633, Z    +0.000, E1   +35.080, E3 -403088.459}
SPL {X  -159.990, Y  +645.423, Z    +0.000, E1   +35.070, E3 -403102.964}
SPL {X  -159.990, Y  +650.555, Z    +0.000, E1   +35.089, E3 -403118.453}
SPL {X  -159.990, Y  +656.270, Z    +0.000, E1   +35.087, E3 -403135.746}
SPL {X  -159.990, Y  +661.105, Z    +0.000, E1   +35.059, E3 -403150.410}
SPL {X  -159.990, Y  +665.311, Z    +0.000, E1   +35.064, E3 -403163.124}
SPL {X  -159.990, Y  +670.193, Z    +0.000, E1   +35.076, E3 -403177.872}
SPL {X  -159.948, Y  +675.148, Z    +0.000, E1   +35.069, E3 -403192.864}
SPL {X  -159.805, Y  +679.202, Z    +0.000, E1   +35.029, E3 -403205.296}
SPL {X  -159.584, Y  +682.885, Z    +0.000, E1   +34.997, E3 -403216.656}
SPL {X  -159.292, Y  +686.426, Z    +0.000, E1   +34.947, E3 -403227.658}
SPL {X  -158.886, Y  +690.264, Z    +0.000, E1   +34.888, E3 -403239.674}
SPL {X  -158.362, Y  +694.266, Z    +0.000, E1   +34.794, E3 -403252.348}
SPL {X  -157.880, Y  +697.401, Z    +0.000, E1   +34.689, E3 -403262.382}
SPL {X  -157.181, Y  +701.346, Z    +0.000, E1   +34.621, E3 -403274.966}
SPL {X  -156.097, Y  +706.580, Z    +0.000, E1   +34.427, E3 -403291.932}
SPL {X  -155.080, Y  +710.833, Z    +0.000, E1   +34.231, E3 -403305.866}
SPL {X  -153.755, Y  +715.731, Z    +0.000, E1   +30.246, E3 -403355.132}
ENDSPLINE

SPLINE
SPL {X  -155.537, Y  +708.983, Z    +0.000, E1   +25.008, E3 -403380.958}
SPL {X  -158.838, Y  +690.666, Z    +0.000, E1   +14.584, E3 -403405.671}
SPL {X  -159.750, Y  +680.262, Z    +0.000, E1    +8.563, E3 -403411.811}
SPL {X  -159.973, Y  +673.798, Z    +0.000, E1    +4.600, E3 -403414.275}
SPL {X  -159.990, Y  +667.448, Z    +0.000, E1    +0.356, E3 -403416.055}
SPL {X  -159.990, Y  +662.686, Z    +0.000, E1    -3.472, E3 -403417.290}
SPL {X  -159.990, Y  +657.071, Z    +0.000, E1    -8.297, E3 -403419.168}
SPL {X  -159.990, Y  +646.193, Z    +0.000, E1   -17.980, E3 -403424.895}
SPL {X  -159.990, Y  +621.124, Z    +0.000, E1   -32.598, E3 -403448.382}
SPL {X  -159.990, Y  +597.855, Z    +0.000, E1   -36.862, E3 -403491.301}
SPL {X  -159.990, Y  +592.884, Z    +0.000, E1   -36.865, E3 -403505.372}
SPL {X  -159.990, Y  +587.104, Z    +0.000, E1   -36.878, E3 -403521.729}
SPL {X  -159.990, Y  +581.795, Z    +0.000, E1   -36.847, E3 -403536.827}
SPL {X  -159.990, Y  +577.286, Z    +0.000, E1   -36.853, E3 -403549.584}
SPL {X  -159.990, Y  +572.409, Z    +0.000, E1   -36.854, E3 -403563.397}
SPL {X  -159.990, Y  +567.110, Z    +0.000, E1   -36.868, E3 -403578.358}
SPL {X  -159.990, Y  +562.387, Z    +0.000, E1   -36.853, E3 -403591.719}
SPL {X  -159.990, Y  +557.944, Z    +0.000, E1   -36.859, E3 -403604.313}
SPL {X  -159.990, Y  +553.661, Z    +0.000, E1   -36.844, E3 -403616.477}
SPL {X  -159.990, Y  +549.195, Z    +0.000, E1   -36.856, E3 -403629.112}
SPL {X  -159.990, Y  +543.458, Z    +0.000, E1   -36.882, E3 -403645.310}
SPL {X  -159.990, Y  +537.639, Z    +0.000, E1   -36.860, E3 -403661.848}
SPL {X  -159.990, Y  +531.894, Z    +0.000, E1   -36.865, E3 -403678.137}
SPL {X  -159.990, Y  +525.940, Z    +0.000, E1   -36.859, E3 -403695.020}
SPL {X  -159.990, Y  +520.301, Z    +0.000, E1   -36.855, E3 -403710.996}
SPL {X  -159.990, Y  +514.308, Z    +0.000, E1   -36.869, E3 -403727.958}
SPL {X  -159.990, Y  +508.591, Z    +0.000, E1   -36.846, E3 -403744.193}
SPL {X  -159.990, Y  +504.505, Z    +0.000, E1   -36.824, E3 -403755.797}
SPL {X  -159.990, Y  +499.829, Z    +0.000, E1   -36.864, E3 -403769.006}
SPL {X  -159.990, Y  +498.054, Z    +0.000, E1   -35.692, E3 -403781.045}
ENDSPLINE

SPLINE
SPL {X  -159.990, Y  +506.994, Z    +0.000, E1   -30.162, E3 -403787.706}
ENDSPLINE

SPLINE
SPL {X  -159.990, Y  +502.084, Z    +0.000, E1   -31.057, E3 -403799.358}
SPL {X  -159.990, Y  +494.586, Z    +0.000, E1   -32.444, E3 -403815.961}
SPL {X  -159.990, Y  +486.073, Z    +0.000, E1   -33.960, E3 -403833.799}
SPL {X  -159.990, Y  +477.314, Z    +0.000, E1   -35.342, E3 -403851.977}
SPL {X  -159.990, Y  +471.459, Z    +0.000, E1   -35.779, E3 -403866.517}
SPL {X  -159.990, Y  +466.474, Z    +0.000, E1   -35.796, E3 -403881.176}
SPL {X  -159.990, Y  +461.990, Z    +0.000, E1   -35.776, E3 -403894.411}
SPL {X  -159.990, Y  +458.524, Z    +0.000, E1   -35.761, E3 -403904.647}
SPL {X  -159.990, Y  +453.597, Z    +0.000, E1   -35.819, E3 -403919.068}
SPL {X  -159.990, Y  +448.227, Z    +0.000, E1   -35.776, E3 -403934.946}
SPL {X  -159.990, Y  +443.707, Z    +0.000, E1   -35.784, E3 -403948.241}
SPL {X  -159.990, Y  +439.109, Z    +0.000, E1   -35.781, E3 -403961.777}
SPL {X  -159.990, Y  +435.535, Z    +0.000, E1   -35.764, E3 -403972.328}
SPL {X  -159.990, Y  +431.100, Z    +0.000, E1   -35.807, E3 -403985.313}
SPL {X  -159.990, Y  +425.407, Z    +0.000, E1   -35.800, E3 -404002.089}
SPL {X  -159.990, Y  +420.199, Z    +0.000, E1   -35.790, E3 -404017.443}
SPL {X  -159.990, Y  +414.514, Z    +0.000, E1   -35.815, E3 -404034.141}
SPL {X  -159.990, Y  +408.600, Z    +0.000, E1   -35.802, E3 -404051.580}
SPL {X  -159.990, Y  +403.496, Z    +0.000, E1   -35.787, E3 -404066.635}
SPL {X  -159.990, Y  +398.606, Z    +0.000, E1   -35.794, E3 -404081.022}
SPL {X  -159.990, Y  +394.138, Z    +0.000, E1   -35.778, E3 -404094.205}
SPL {X  -159.990, Y  +390.065, Z    +0.000, E1   -35.780, E3 -404106.196}
SPL {X  -159.990, Y  +385.506, Z    +0.000, E1   -35.789, E3 -404119.601}
SPL {X  -159.976, Y  +380.359, Z    +0.000, E1   -35.797, E3 -404134.750}
SPL {X  -159.831, Y  +375.358, Z    +0.000, E1   -35.763, E3 -404149.640}
SPL {X  -159.547, Y  +370.604, Z    +0.000, E1   -35.724, E3 -404163.940}
SPL {X  -159.134, Y  +365.969, Z    +0.000, E1   -35.644, E3 -404178.026}
SPL {X  -158.606, Y  +361.498, Z    +0.000, E1   -35.550, E3 -404191.790}
SPL {X  -157.918, Y  +356.833, Z    +0.000, E1   -35.439, E3 -404206.243}
SPL {X  -157.185, Y  +352.671, Z    +0.000, E1   -35.292, E3 -404219.303}
SPL {X  -156.302, Y  +348.345, Z    +0.000, E1   -35.165, E3 -404232.924}
SPL {X  -155.054, Y  +343.066, Z    +0.000, E1   -34.964, E3 -404249.739}
SPL {X  -154.305, Y  +340.232, Z    +0.000, E1   -28.975, E3 -404307.299}
ENDSPLINE

SPLINE
SPL {X  -158.456, Y  +360.399, Z    +0.000, E1   -16.490, E3 -404344.119}
SPL {X  -159.553, Y  +370.677, Z    +0.000, E1   -10.576, E3 -404351.879}
SPL {X  -159.960, Y  +379.402, Z    +0.000, E1    -5.303, E3 -404355.899}
SPL {X  -159.990, Y  +385.983, Z    +0.000, E1    -0.882, E3 -404357.971}
SPL {X  -159.990, Y  +390.933, Z    +0.000, E1    +2.877, E3 -404359.419}
SPL {X  -159.990, Y  +396.375, Z    +0.000, E1    +7.538, E3 -404361.194}
SPL {X  -159.990, Y  +404.277, Z    +0.000, E1   +14.543, E3 -404364.857}
SPL {X  -159.990, Y  +423.101, Z    +0.000, E1   +27.351, E3 -404381.296}
SPL {X  -159.990, Y  +430.933, Z    +0.000, E1   +30.672, E3 -404391.267}
SPL {X  -159.990, Y  +452.779, Z    +0.000, E1   +35.077, E3 -404433.430}
SPL {X  -159.990, Y  +457.209, Z    +0.000, E1   +35.039, E3 -404446.890}
SPL {X  -159.990, Y  +460.708, Z    +0.000, E1   +35.045, E3 -404457.472}
SPL {X  -159.990, Y  +464.162, Z    +0.000, E1   +35.038, E3 -404467.928}
SPL {X  -159.990, Y  +467.857, Z    +0.000, E1   +35.053, E3 -404479.085}
SPL {X  -159.990, Y  +471.326, Z    +0.000, E1   +35.038, E3 -404489.580}
SPL {X  -159.990, Y  +474.610, Z    +0.000, E1   +35.053, E3 -404499.480}
SPL {X  -159.990, Y  +478.303, Z    +0.000, E1   +35.049, E3 -404510.652}
SPL {X  -159.990, Y  +482.537, Z    +0.000, E1   +35.066, E3 -404523.443}
SPL {X  -159.990, Y  +487.181, Z    +0.000, E1   +35.054, E3 -404537.526}
SPL {X  -159.990, Y  +492.368, Z    +0.000, E1   +35.076, E3 -404553.198}
SPL {X  -159.990, Y  +497.072, Z    +0.000, E1   +35.040, E3 -404567.494}
SPL {X  -159.990, Y  +501.645, Z    +0.000, E1   +35.067, E3 -404581.277}
SPL {X  -159.990, Y  +506.307, Z    +0.000, E1   +35.049, E3 -404595.399}
SPL {X  -159.990, Y  +511.643, Z    +0.000, E1   +35.091, E3 -404611.479}
SPL {X  -159.990, Y  +517.156, Z    +0.000, E1   +35.059, E3 -404628.198}
SPL {X  -159.990, Y  +521.637, Z    +0.000, E1   +35.056, E3 -404641.761}
SPL {X  -159.990, Y  +526.246, Z    +0.000, E1   +35.065, E3 -404655.664}
SPL {X  -159.990, Y  +530.289, Z    +0.000, E1   +35.044, E3 -404667.951}
SPL {X  -159.990, Y  +534.797, Z    +0.000, E1   +35.069, E3 -404681.551}
SPL {X  -159.990, Y  +538.710, Z    +0.000, E1   +35.033, E3 -404693.448}
SPL {X  -159.990, Y  +542.114, Z    +0.000, E1   +35.053, E3 -404703.700}
SPL {X  -159.990, Y  +546.612, Z    +0.000, E1   +35.065, E3 -404717.271}
SPL {X  -159.990, Y  +551.596, Z    +0.000, E1   +35.079, E3 -404732.306}
SPL {X  -159.990, Y  +556.051, Z    +0.000, E1   +35.060, E3 -404745.769}
SPL {X  -159.990, Y  +560.931, Z    +0.000, E1   +35.098, E3 -404760.474}
SPL {X  -159.990, Y  +564.815, Z    +0.000, E1   +35.041, E3 -404772.322}
SPL {X  -159.990, Y  +567.494, Z    +0.000, E1   +35.052, E3 -404780.402}
SPL {X  -159.990, Y  +571.374, Z    +0.000, E1   +35.070, E3 -404792.105}
SPL {X  -159.990, Y  +575.771, Z    +0.000, E1   +35.064, E3 -404805.410}
SPL {X  -159.990, Y  +580.750, Z    +0.000, E1   +35.087, E3 -404820.433}
SPL {X  -159.990, Y  +585.414, Z    +0.000, E1   +35.059, E3 -404834.579}
SPL {X  -159.990, Y  +590.166, Z    +0.000, E1   +35.084, E3 -404848.907}
SPL {X  -159.990, Y  +595.313, Z    +0.000, E1   +35.073, E3 -404864.486}
SPL {X  -159.990, Y  +599.479, Z    +0.000, E1   +35.059, E3 -404877.104}
SPL {X  -159.990, Y  +603.289, Z    +0.000, E1   +35.068, E3 -404888.593}
SPL {X  -159.990, Y  +607.919, Z    +0.000, E1   +35.079, E3 -404902.582}
SPL {X  -159.990, Y  +613.036, Z    +0.000, E1   +35.082, E3 -404918.052}
SPL {X  -159.990, Y  +617.577, Z    +0.000, E1   +35.061, E3 -404931.814}
SPL {X  -159.990, Y  +621.534, Z    +0.000, E1   +35.068, E3 -404943.748}
SPL {X  -159.990, Y  +626.426, Z    +0.000, E1   +35.093, E3 -404958.507}
SPL {X  -159.990, Y  +631.553, Z    +0.000, E1   +35.068, E3 -404974.065}
SPL {X  -159.990, Y  +635.965, Z    +0.000, E1   +35.065, E3 -404987.414}
SPL {X  -159.990, Y  +640.633, Z    +0.000, E1   +35.080, E3 -405001.502}
SPL {X  -159.990, Y  +645.423, Z    +0.000, E1   +35.070, E3 -405016.007}
SPL {X  -159.990, Y  +650.555, Z    +0.000, E1   +35.089, E3 -405031.497}
SPL {X  -159.990, Y  +656.270, Z    +0.000, E1   +35.087, E3 -405048.790}
SPL {X  -159.990, Y  +661.105, Z    +0.000, E1   +35.059, E3 -405063.453}
SPL {X  -159.990, Y  +665.311, Z    +0.000, E1   +35.064, E3 -405076.168}
SPL {X  -159.990, Y  +668.650, Z    +0.000, E1   +35.040, E3 -405086.308}
SPL {X  -159.990, Y  +671.288, Z    +0.000, E1   +35.046, E3 -405094.272}
SPL {X  -159.948, Y  +675.148, Z    +0.000, E1   +35.069, E3 -405105.907}
SPL {X  -159.752, Y  +680.228, Z    +0.000, E1   +35.050, E3 -405121.455}
SPL {X  -159.371, Y  +685.563, Z    +0.000, E1   +34.989, E3 -405137.966}
SPL {X  -158.886, Y  +690.264, Z    +0.000, E1   +34.888, E3 -405152.718}
SPL {X  -158.362, Y  +694.266, Z    +0.000, E1   +34.794, E3 -405165.391}
SPL {X  -157.614, Y  +698.973, Z    +0.000, E1   +34.690, E3 -405180.392}
SPL {X  -156.901, Y  +702.787, Z    +0.000, E1   +34.523, E3 -405192.735}
SPL {X  -156.097, Y  +706.580, Z    +0.000, E1   +34.427, E3 -405204.975}
SPL {X  -155.080, Y  +710.833, Z    +0.000, E1   +34.231, E3 -405218.909}
SPL {X  -153.755, Y  +715.731, Z    +0.000, E1   +30.246, E3 -405268.175}
ENDSPLINE

SPLINE
SPL {X  -155.537, Y  +708.983, Z    +0.000, E1   +25.008, E3 -405294.002}
SPL {X  -158.838, Y  +690.666, Z    +0.000, E1   +14.584, E3 -405318.714}
SPL {X  -159.750, Y  +680.262, Z    +0.000, E1    +8.563, E3 -405324.855}
SPL {X  -159.973, Y  +673.798, Z    +0.000, E1    +4.600, E3 -405327.319}
SPL {X  -159.990, Y  +668.863, Z    +0.000, E1    +1.298, E3 -405328.758}
SPL {X  -159.990, Y  +663.839, Z    +0.000, E1    -2.454, E3 -405330.019}
SPL {X  -159.990, Y  +658.349, Z    +0.000, E1    -7.223, E3 -405331.701}
SPL {X  -159.990, Y  +653.910, Z    +0.000, E1   -11.344, E3 -405333.469}
SPL {X  -159.990, Y  +646.193, Z    +0.000, E1   -17.980, E3 -405337.938}
SPL {X  -159.990, Y  +621.124, Z    +0.000, E1   -32.598, E3 -405361.425}
SPL {X  -159.990, Y  +599.888, Z    +0.000, E1   -36.828, E3 -405398.665}
SPL {X  -159.990, Y  +595.346, Z    +0.000, E1   -36.880, E3 -405411.431}
SPL {X  -159.990, Y  +589.749, Z    +0.000, E1   -36.860, E3 -405427.304}
SPL {X  -159.990, Y  +585.754, Z    +0.000, E1   -36.838, E3 -405438.659}
SPL {X  -159.990, Y  +581.795, Z    +0.000, E1   -36.847, E3 -405449.871}
SPL {X  -159.990, Y  +577.286, Z    +0.000, E1   -36.853, E3 -405462.628}
SPL {X  -159.990, Y  +572.409, Z    +0.000, E1   -36.854, E3 -405476.440}
SPL {X  -159.990, Y  +567.110, Z    +0.000, E1   -36.868, E3 -405491.401}
SPL {X  -159.990, Y  +562.387, Z    +0.000, E1   -36.853, E3 -405504.763}
SPL {X  -159.990, Y  +557.944, Z    +0.000, E1   -36.859, E3 -405517.356}
SPL {X  -159.990, Y  +552.571, Z    +0.000, E1   -36.873, E3 -405532.560}
SPL {X  -159.990, Y  +548.223, Z    +0.000, E1   -36.832, E3 -405544.951}
SPL {X  -159.990, Y  +543.458, Z    +0.000, E1   -36.882, E3 -405558.353}
SPL {X  -159.990, Y  +537.639, Z    +0.000, E1   -36.860, E3 -405574.891}
SPL {X  -159.990, Y  +531.894, Z    +0.000, E1   -36.865, E3 -405591.180}
SPL {X  -159.990, Y  +525.940, Z    +0.000, E1   -36.859, E3 -405608.063}
SPL {X  -159.990, Y  +520.301, Z    +0.000, E1   -36.855, E3 -405624.039}
SPL {X  -159.990, Y  +516.005, Z    +0.000, E1   -36.824, E3 -405636.266}
SPL {X  -159.990, Y  +511.408, Z    +0.000, E1   -36.858, E3 -405649.235}
SPL {X  -159.990, Y  +505.756, Z    +0.000, E1   -36.857, E3 -405665.244}
SPL {X  -159.990, Y  +499.829, Z    +0.000, E1   -36.864, E3 -405682.049}
SPL {X  -159.990, Y  +498.054, Z    +0.000, E1   -35.692, E3 -405694.088}
ENDSPLINE

SPLINE
SPL {X  -159.990, Y  +506.994, Z    +0.000, E1   -30.162, E3 -405700.750}
ENDSPLINE

SPLINE
SPL {X  -159.990, Y  +502.084, Z    +0.000, E1   -31.057, E3 -405712.401}
SPL {X  -159.990, Y  +494.586, Z    +0.000, E1   -32.444, E3 -405729.005}
SPL {X  -159.990, Y  +486.073, Z    +0.000, E1   -33.960, E3 -405746.842}
SPL {X  -159.990, Y  +477.314, Z    +0.000, E1   -35.342, E3 -405765.021}
SPL {X  -159.990, Y  +471.459, Z    +0.000, E1   -35.779, E3 -405779.560}
SPL {X  -159.990, Y  +467.485, Z    +0.000, E1   -35.768, E3 -405791.290}
SPL {X  -159.990, Y  +462.739, Z    +0.000, E1   -35.799, E3 -405805.218}
SPL {X  -159.990, Y  +457.385, Z    +0.000, E1   -35.788, E3 -405821.001}
SPL {X  -159.990, Y  +452.637, Z    +0.000, E1   -35.783, E3 -405834.993}
SPL {X  -159.990, Y  +448.227, Z    +0.000, E1   -35.776, E3 -405847.989}
SPL {X  -159.990, Y  +443.707, Z    +0.000, E1   -35.784, E3 -405861.285}
SPL {X  -159.990, Y  +439.109, Z    +0.000, E1   -35.781, E3 -405874.821}
SPL {X  -159.990, Y  +434.400, Z    +0.000, E1   -35.789, E3 -405888.675}
SPL {X  -159.990, Y  +430.115, Z    +0.000, E1   -35.777, E3 -405901.292}
SPL {X  -159.990, Y  +425.407, Z    +0.000, E1   -35.800, E3 -405915.132}
SPL {X  -159.990, Y  +420.199, Z    +0.000, E1   -35.790, E3 -405930.486}
SPL {X  -159.990, Y  +414.514, Z    +0.000, E1   -35.815, E3 -405947.185}
SPL {X  -159.990, Y  +408.600, Z    +0.000, E1   -35.802, E3 -405964.624}
SPL {X  -159.990, Y  +403.496, Z    +0.000, E1   -35.787, E3 -405979.678}
SPL {X  -159.990, Y  +398.606, Z    +0.000, E1   -35.794, E3 -405994.066}
SPL {X  -159.990, Y  +394.138, Z    +0.000, E1   -35.778, E3 -406007.249}
SPL {X  -159.990, Y  +388.813, Z    +0.000, E1   -35.819, E3 -406022.861}
SPL {X  -159.990, Y  +383.172, Z    +0.000, E1   -35.789, E3 -406039.515}
SPL {X  -159.936, Y  +378.352, Z    +0.000, E1   -35.782, E3 -406053.754}
SPL {X  -159.693, Y  +372.749, Z    +0.000, E1   -35.767, E3 -406070.486}
SPL {X  -159.203, Y  +366.647, Z    +0.000, E1   -35.680, E3 -406088.972}
SPL {X  -158.715, Y  +362.338, Z    +0.000, E1   -35.547, E3 -406102.277}
SPL {X  -158.237, Y  +358.884, Z    +0.000, E1   -35.480, E3 -406112.934}
SPL {X  -157.724, Y  +355.670, Z    +0.000, E1   -35.371, E3 -406122.968}
SPL {X  -157.185, Y  +352.671, Z    +0.000, E1   -35.292, E3 -406132.347}
SPL {X  -156.302, Y  +348.345, Z    +0.000, E1   -35.165, E3 -406145.968}
SPL {X  -155.054, Y  +343.066, Z    +0.000, E1   -34.964, E3 -406162.783}
SPL {X  -154.305, Y  +340.232, Z    +0.000, E1   -28.975, E3 -406220.342}
ENDSPLINE

SPLINE
SPL {X  -158.456, Y  +360.399, Z    +0.000, E1   -16.490, E3 -406257.162}
SPL {X  -159.553, Y  +370.677, Z    +0.000, E1   -10.576, E3 -406264.922}
SPL {X  -159.960, Y  +379.402, Z    +0.000, E1    -5.303, E3 -406268.942}
SPL {X  -159.990, Y  +387.301, Z    +0.000, E1    -0.001, E3 -406271.404}
SPL {X  -159.990, Y  +392.161, Z    +0.000, E1    +3.946, E3 -406272.815}
SPL {X  -159.990, Y  +396.375, Z    +0.000, E1    +7.538, E3 -406274.238}
SPL {X  -159.990, Y  +404.277, Z    +0.000, E1   +14.543, E3 -406277.901}
SPL {X  -159.990, Y  +423.101, Z    +0.000, E1   +27.351, E3 -406294.339}
SPL {X  -159.990, Y  +430.933, Z    +0.000, E1   +30.672, E3 -406304.310}
SPL {X  -159.990, Y  +451.842, Z    +0.000, E1   +35.050, E3 -406343.682}
SPL {X  -159.990, Y  +456.402, Z    +0.000, E1   +35.061, E3 -406357.458}
SPL {X  -159.990, Y  +460.708, Z    +0.000, E1   +35.045, E3 -406370.515}
SPL {X  -159.990, Y  +464.162, Z    +0.000, E1   +35.038, E3 -406380.972}
SPL {X  -159.990, Y  +467.857, Z    +0.000, E1   +35.053, E3 -406392.129}
SPL {X  -159.990, Y  +471.326, Z    +0.000, E1   +35.038, E3 -406402.624}
SPL {X  -159.990, Y  +474.610, Z    +0.000, E1   +35.053, E3 -406412.523}
SPL {X  -159.990, Y  +478.303, Z    +0.000, E1   +35.049, E3 -406423.696}
SPL {X  -159.990, Y  +482.537, Z    +0.000, E1   +35.066, E3 -406436.487}
SPL {X  -159.990, Y  +487.181, Z    +0.000, E1   +35.054, E3 -406450.570}
SPL {X  -159.990, Y  +490.807, Z    +0.000, E1   +35.036, E3 -406461.571}
SPL {X  -159.990, Y  +493.669, Z    +0.000, E1   +35.034, E3 -406470.250}
SPL {X  -159.990, Y  +497.072, Z    +0.000, E1   +35.040, E3 -406480.538}
SPL {X  -159.990, Y  +501.645, Z    +0.000, E1   +35.067, E3 -406494.321}
SPL {X  -159.990, Y  +507.359, Z    +0.000, E1   +35.080, E3 -406511.578}
SPL {X  -159.990, Y  +512.562, Z    +0.000, E1   +35.055, E3 -406527.360}
SPL {X  -159.990, Y  +517.156, Z    +0.000, E1   +35.059, E3 -406541.241}
SPL {X  -159.990, Y  +521.637, Z    +0.000, E1   +35.056, E3 -406554.804}
SPL {X  -159.990, Y  +525.227, Z    +0.000, E1   +35.041, E3 -406565.665}
SPL {X  -159.990, Y  +529.413, Z    +0.000, E1   +35.072, E3 -406578.294}
SPL {X  -159.990, Y  +534.797, Z    +0.000, E1   +35.069, E3 -406594.594}
SPL {X  -159.990, Y  +538.710, Z    +0.000, E1   +35.033, E3 -406606.491}
SPL {X  -159.990, Y  +542.114, Z    +0.000, E1   +35.053, E3 -406616.743}
SPL {X  -159.990, Y  +546.612, Z    +0.000, E1   +35.065, E3 -406630.315}
SPL {X  -159.990, Y  +551.596, Z    +0.000, E1   +35.079, E3 -406645.350}
SPL {X  -159.990, Y  +557.043, Z    +0.000, E1   +35.087, E3 -406661.772}
SPL {X  -159.990, Y  +562.842, Z    +0.000, E1   +35.098, E3 -406679.304}
SPL {X  -159.990, Y  +568.750, Z    +0.000, E1   +35.087, E3 -406697.190}
SPL {X  -159.990, Y  +574.780, Z    +0.000, E1   +35.101, E3 -406715.401}
SPL {X  -159.990, Y  +580.750, Z    +0.000, E1   +35.087, E3 -406733.476}
SPL {X  -159.990, Y  +585.414, Z    +0.000, E1   +35.059, E3 -406747.623}
SPL {X  -159.990, Y  +588.716, Z    +0.000, E1   +35.047, E3 -406757.625}
SPL {X  -159.990, Y  +592.923, Z    +0.000, E1   +35.084, E3 -406770.290}
SPL {X  -159.990, Y  +598.554, Z    +0.000, E1   +35.088, E3 -406787.309}
SPL {X  -159.990, Y  +603.289, Z    +0.000, E1   +35.068, E3 -406801.636}
SPL {X  -159.990, Y  +607.919, Z    +0.000, E1   +35.079, E3 -406815.625}
SPL {X  -159.990, Y  +613.036, Z    +0.000, E1   +35.082, E3 -406831.096}
SPL {X  -159.990, Y  +617.577, Z    +0.000, E1   +35.061, E3 -406844.857}
SPL {X  -159.990, Y  +621.534, Z    +0.000, E1   +35.068, E3 -406856.791}
SPL {X  -159.990, Y  +626.426, Z    +0.000, E1   +35.093, E3 -406871.551}
SPL {X  -159.990, Y  +631.553, Z    +0.000, E1   +35.068, E3 -406887.109}
SPL {X  -159.990, Y  +636.917, Z    +0.000, E1   +35.095, E3 -406903.288}
SPL {X  -159.990, Y  +641.534, Z    +0.000, E1   +35.053, E3 -406917.316}
SPL {X  -159.990, Y  +646.430, Z    +0.000, E1   +35.102, E3 -406932.047}
SPL {X  -159.990, Y  +651.502, Z    +0.000, E1   +35.058, E3 -406947.457}
SPL {X  -159.990, Y  +654.793, Z    +0.000, E1   +35.049, E3 -406957.420}
SPL {X  -159.990, Y  +657.535, Z    +0.000, E1   +35.049, E3 -406965.717}
SPL {X  -159.990, Y  +661.105, Z    +0.000, E1   +35.059, E3 -406976.497}
SPL {X  -159.990, Y  +665.311, Z    +0.000, E1   +35.064, E3 -406989.211}
SPL {X  -159.990, Y  +670.193, Z    +0.000, E1   +35.076, E3 -407003.959}
SPL {X  -159.948, Y  +675.148, Z    +0.000, E1   +35.069, E3 -407018.951}
SPL {X  -159.752, Y  +680.228, Z    +0.000, E1   +35.050, E3 -407034.498}
SPL {X  -159.371, Y  +685.563, Z    +0.000, E1   +34.989, E3 -407051.010}
SPL {X  -158.886, Y  +690.264, Z    +0.000, E1   +34.888, E3 -407065.761}
SPL {X  -158.362, Y  +694.266, Z    +0.000, E1   +34.794, E3 -407078.435}
SPL {X  -157.614, Y  +698.973, Z    +0.000, E1   +34.690, E3 -407093.435}
SPL {X  -156.640, Y  +704.066, Z    +0.000, E1   +34.516, E3 -407109.861}
SPL {X  -155.835, Y  +707.723, Z    +0.000, E1   +34.344, E3 -407121.803}
SPL {X  -155.080, Y  +710.833, Z    +0.000, E1   +34.231, E3 -407131.953}
SPL {X  -153.755, Y  +715.731, Z    +0.000, E1   +30.246, E3 -407181.219}
ENDSPLINE

SPLINE
SPL {X  -155.537, Y  +708.983, Z    +0.000, E1   +25.008, E3 -407207.045}
SPL {X  -158.838, Y  +690.666, Z    +0.000, E1   +14.584, E3 -407231.758}
SPL {X  -159.750, Y  +680.262, Z    +0.000, E1    +8.563, E3 -407237.898}
SPL {X  -159.973, Y  +673.798, Z    +0.000, E1    +4.600, E3 -407240.362}
SPL {X  -159.990, Y  +668.863, Z    +0.000, E1    +1.298, E3 -407241.802}
SPL {X  -159.990, Y  +663.839, Z    +0.000, E1    -2.454, E3 -407243.062}
SPL {X  -159.990, Y  +657.071, Z    +0.000, E1    -8.297, E3 -407245.255}
SPL {X  -159.990, Y  +646.193, Z    +0.000, E1   -17.980, E3 -407250.982}
SPL {X  -159.990, Y  +621.124, Z    +0.000, E1   -32.598, E3 -407274.469}
SPL {X  -159.990, Y  +597.855, Z    +0.000, E1   -36.862, E3 -407317.388}
SPL {X  -159.990, Y  +592.884, Z    +0.000, E1   -36.865, E3 -407331.459}
SPL {X  -159.990, Y  +587.104, Z    +0.000, E1   -36.878, E3 -407347.816}
SPL {X  -159.990, Y  +581.795, Z    +0.000, E1   -36.847, E3 -407362.914}
SPL {X  -159.990, Y  +577.286, Z    +0.000, E1   -36.853, E3 -407375.671}
SPL {X  -159.990, Y  +572.409, Z    +0.000, E1   -36.854, E3 -407389.484}
SPL {X  -159.990, Y  +567.110, Z    +0.000, E1   -36.868, E3 -407404.445}
SPL {X  -159.990, Y  +562.387, Z    +0.000, E1   -36.853, E3 -407417.806}
SPL {X  -159.990, Y  +557.944, Z    +0.000, E1   -36.859, E3 -407430.400}
SPL {X  -159.990, Y  +553.661, Z    +0.000, E1   -36.844, E3 -407442.564}
SPL {X  -159.990, Y  +549.195, Z    +0.000, E1   -36.856, E3 -407455.199}
SPL {X  -159.990, Y  +544.733, Z    +0.000, E1   -36.845, E3 -407467.845}
SPL {X  -159.990, Y  +539.889, Z    +0.000, E1   -36.872, E3 -407481.529}
SPL {X  -159.990, Y  +534.469, Z    +0.000, E1   -36.855, E3 -407496.927}
SPL {X  -159.990, Y  +528.569, Z    +0.000, E1   -36.871, E3 -407513.645}
SPL {X  -159.990, Y  +522.641, Z    +0.000, E1   -36.854, E3 -407530.456}
SPL {X  -159.990, Y  +517.225, Z    +0.000, E1   -36.859, E3 -407545.790}
SPL {X  -159.990, Y  +512.789, Z    +0.000, E1   -36.824, E3 -407558.417}
SPL {X  -159.990, Y  +508.591, Z    +0.000, E1   -36.846, E3 -407570.280}
SPL {X  -159.990, Y  +503.454, Z    +0.000, E1   -36.847, E3 -407584.835}
SPL {X  -159.990, Y  +498.817, Z    +0.000, E1   -36.830, E3 -407598.018}
SPL {X  -159.990, Y  +498.054, Z    +0.000, E1   -35.692, E3 -407607.132}
ENDSPLINE

SPLINE
SPL {X  -159.990, Y  +506.994, Z    +0.000, E1   -30.162, E3 -407613.793}
ENDSPLINE

SPLINE
SPL {X  -159.990, Y  +502.084, Z    +0.000, E1   -31.057, E3 -407625.445}
SPL {X  -159.990, Y  +494.586, Z    +0.000, E1   -32.444, E3 -407642.048}
SPL {X  -159.990, Y  +487.723, Z    +0.000, E1   -33.658, E3 -407656.501}
SPL {X  -159.990, Y  +481.374, Z    +0.000, E1   -34.706, E3 -407669.705}
SPL {X  -159.990, Y  +475.503, Z    +0.000, E1   -35.597, E3 -407681.757}
SPL {X  -159.990, Y  +471.459, Z    +0.000, E1   -35.779, E3 -407692.604}
SPL {X  -159.990, Y  +466.474, Z    +0.000, E1   -35.796, E3 -407707.262}
SPL {X  -159.990, Y  +461.990, Z    +0.000, E1   -35.776, E3 -407720.498}
SPL {X  -159.990, Y  +457.385, Z    +0.000, E1   -35.788, E3 -407734.045}
SPL {X  -159.990, Y  +452.637, Z    +0.000, E1   -35.783, E3 -407748.036}
SPL {X  -159.990, Y  +446.982, Z    +0.000, E1   -35.815, E3 -407764.638}
SPL {X  -159.990, Y  +442.593, Z    +0.000, E1   -35.759, E3 -407777.647}
SPL {X  -159.990, Y  +439.109, Z    +0.000, E1   -35.781, E3 -407787.864}
SPL {X  -159.990, Y  +435.535, Z    +0.000, E1   -35.764, E3 -407798.415}
SPL {X  -159.990, Y  +431.100, Z    +0.000, E1   -35.807, E3 -407811.400}
SPL {X  -159.990, Y  +426.641, Z    +0.000, E1   -35.769, E3 -407824.587}
SPL {X  -159.990, Y  +422.627, Z    +0.000, E1   -35.788, E3 -407836.384}
SPL {X  -159.990, Y  +417.866, Z    +0.000, E1   -35.788, E3 -407850.398}
SPL {X  -159.990, Y  +413.498, Z    +0.000, E1   -35.779, E3 -407863.279}
SPL {X  -159.990, Y  +408.600, Z    +0.000, E1   -35.802, E3 -407877.667}
SPL {X  -159.990, Y  +403.496, Z    +0.000, E1   -35.787, E3 -407892.722}
SPL {X  -159.990, Y  +398.606, Z    +0.000, E1   -35.794, E3 -407907.109}
SPL {X  -159.990, Y  +394.138, Z    +0.000, E1   -35.778, E3 -407920.292}
SPL {X  -159.990, Y  +388.813, Z    +0.000, E1   -35.819, E3 -407935.905}
SPL {X  -159.990, Y  +383.172, Z    +0.000, E1   -35.789, E3 -407952.559}
SPL {X  -159.957, Y  +379.262, Z    +0.000, E1   -35.764, E3 -407964.130}
SPL {X  -159.831, Y  +375.358, Z    +0.000, E1   -35.763, E3 -407975.727}
SPL {X  -159.547, Y  +370.604, Z    +0.000, E1   -35.724, E3 -407990.027}
SPL {X  -159.134, Y  +365.969, Z    +0.000, E1   -35.644, E3 -408004.112}
SPL {X  -158.715, Y  +362.338, Z    +0.000, E1   -35.547, E3 -408015.321}
SPL {X  -158.237, Y  +358.884, Z    +0.000, E1   -35.480, E3 -408025.977}
SPL {X  -157.724, Y  +355.670, Z    +0.000, E1   -35.371, E3 -408036.012}
SPL {X  -157.185, Y  +352.671, Z    +0.000, E1   -35.292, E3 -408045.390}
SPL {X  -156.582, Y  +349.653, Z    +0.000, E1   -35.175, E3 -408054.924}
SPL {X  -155.743, Y  +345.880, Z    +0.000, E1   -35.068, E3 -408066.851}
SPL {X  -154.759, Y  +341.925, Z    +0.000, E1   -34.868, E3 -408079.557}
SPL {X  -154.305, Y  +340.232, Z    +0.000, E1   -28.975, E3 -408133.386}
ENDSPLINE

SPLINE
SPL {X  -158.456, Y  +360.399, Z    +0.000, E1   -16.490, E3 -408170.206}
SPL {X  -159.553, Y  +370.677, Z    +0.000, E1   -10.576, E3 -408177.966}
SPL {X  -159.960, Y  +379.402, Z    +0.000, E1    -5.303, E3 -408181.986}
SPL {X  -159.990, Y  +385.983, Z    +0.000, E1    -0.882, E3 -408184.058}
SPL {X  -159.990, Y  +390.933, Z    +0.000, E1    +2.877, E3 -408185.506}
SPL {X  -159.990, Y  +396.375, Z    +0.000, E1    +7.538, E3 -408187.281}
SPL {X  -159.990, Y  +405.219, Z    +0.000, E1   +15.296, E3 -408191.599}
SPL {X  -159.990, Y  +427.882, Z    +0.000, E1   +29.477, E3 -408213.278}
SPL {X  -159.990, Y  +451.842, Z    +0.000, E1   +35.050, E3 -408256.725}
SPL {X  -159.990, Y  +456.402, Z    +0.000, E1   +35.061, E3 -408270.501}
SPL {X  -159.990, Y  +460.708, Z    +0.000, E1   +35.045, E3 -408283.559}
SPL {X  -159.990, Y  +465.240, Z    +0.000, E1   +35.066, E3 -408297.235}
SPL {X  -159.990, Y  +470.278, Z    +0.000, E1   +35.063, E3 -408312.468}
SPL {X  -159.990, Y  +474.610, Z    +0.000, E1   +35.053, E3 -408325.567}
SPL {X  -159.990, Y  +478.303, Z    +0.000, E1   +35.049, E3 -408336.739}
SPL {X  -159.990, Y  +482.537, Z    +0.000, E1   +35.066, E3 -408349.530}
SPL {X  -159.990, Y  +487.181, Z    +0.000, E1   +35.054, E3 -408363.613}
SPL {X  -159.990, Y  +490.807, Z    +0.000, E1   +35.036, E3 -408374.614}
SPL {X  -159.990, Y  +493.669, Z    +0.000, E1   +35.034, E3 -408383.294}
SPL {X  -159.990, Y  +497.072, Z    +0.000, E1   +35.040, E3 -408393.581}
SPL {X  -159.990, Y  +501.645, Z    +0.000, E1   +35.067, E3 -408407.364}
SPL {X  -159.990, Y  +506.307, Z    +0.000, E1   +35.049, E3 -408421.486}
SPL {X  -159.990, Y  +510.443, Z    +0.000, E1   +35.051, E3 -408433.999}
SPL {X  -159.990, Y  +514.632, Z    +0.000, E1   +35.050, E3 -408446.669}
SPL {X  -159.990, Y  +518.055, Z    +0.000, E1   +35.037, E3 -408457.038}
SPL {X  -159.990, Y  +521.637, Z    +0.000, E1   +35.056, E3 -408467.848}
SPL {X  -159.990, Y  +526.246, Z    +0.000, E1   +35.065, E3 -408481.751}
SPL {X  -159.990, Y  +530.289, Z    +0.000, E1   +35.044, E3 -408494.037}
SPL {X  -159.990, Y  +534.797, Z    +0.000, E1   +35.069, E3 -408507.638}
SPL {X  -159.990, Y  +538.710, Z    +0.000, E1   +35.033, E3 -408519.535}
SPL {X  -159.990, Y  +542.114, Z    +0.000, E1   +35.053, E3 -408529.787}
SPL {X  -159.990, Y  +545.724, Z    +0.000, E1   +35.043, E3 -408540.711}
SPL {X  -159.990, Y  +549.546, Z    +0.000, E1   +35.061, E3 -408552.236}
SPL {X  -159.990, Y  +552.868, Z    +0.000, E1   +35.047, E3 -408562.278}
SPL {X  -159.990, Y  +557.043, Z    +0.000, E1   +35.087, E3 -408574.815}
SPL {X  -159.990, Y  +561.808, Z    +0.000, E1   +35.066, E3 -408589.268}
SPL {X  -159.990, Y  +566.542, Z    +0.000, E1   +35.080, E3 -408603.568}
SPL {X  -159.990, Y  +570.261, Z    +0.000, E1   +35.046, E3 -408614.864}
SPL {X  -159.990, Y  +574.780, Z    +0.000, E1   +35.101, E3 -408628.444}
SPL {X  -159.990, Y  +579.185, Z    +0.000, E1   +35.047, E3 -408641.845}
SPL {X  -159.990, Y  +581.944, Z    +0.000, E1   +35.051, E3 -408650.184}
SPL {X  -159.990, Y  +585.414, Z    +0.000, E1   +35.059, E3 -408660.666}
SPL {X  -159.990, Y  +588.716, Z    +0.000, E1   +35.047, E3 -408670.669}
SPL {X  -159.990, Y  +592.923, Z    +0.000, E1   +35.084, E3 -408683.333}
SPL {X  -159.990, Y  +598.554, Z    +0.000, E1   +35.088, E3 -408700.352}
SPL {X  -159.990, Y  +603.289, Z    +0.000, E1   +35.068, E3 -408714.680}
SPL {X  -159.990, Y  +607.919, Z    +0.000, E1   +35.079, E3 -408728.668}
SPL {X  -159.990, Y  +613.036, Z    +0.000, E1   +35.082, E3 -408744.139}
SPL {X  -159.990, Y  +617.577, Z    +0.000, E1   +35.061, E3 -408757.901}
SPL {X  -159.990, Y  +621.534, Z    +0.000, E1   +35.068, E3 -408769.835}
SPL {X  -159.990, Y  +626.426, Z    +0.000, E1   +35.093, E3 -408784.594}
SPL {X  -159.990, Y  +631.553, Z    +0.000, E1   +35.068, E3 -408800.152}
SPL {X  -159.990, Y  +635.965, Z    +0.000, E1   +35.065, E3 -408813.501}
SPL {X  -159.990, Y  +640.633, Z    +0.000, E1   +35.080, E3 -408827.589}
SPL {X  -159.990, Y  +645.423, Z    +0.000, E1   +35.070, E3 -408842.094}
SPL {X  -159.990, Y  +650.555, Z    +0.000, E1   +35.089, E3 -408857.584}
SPL {X  -159.990, Y  +656.270, Z    +0.000, E1   +35.087, E3 -408874.876}
SPL {X  -159.990, Y  +661.105, Z    +0.000, E1   +35.059, E3 -408889.540}
SPL {X  -159.990, Y  +665.311, Z    +0.000, E1   +35.064, E3 -408902.255}
SPL {X  -159.990, Y  +670.193, Z    +0.000, E1   +35.076, E3 -408917.002}
SPL {X  -159.948, Y  +675.148, Z    +0.000, E1   +35.069, E3 -408931.994}
SPL {X  -159.805, Y  +679.202, Z    +0.000, E1   +35.029, E3 -408944.426}
SPL {X  -159.584, Y  +682.885, Z    +0.000, E1   +34.997, E3 -408955.786}
SPL {X  -159.292, Y  +686.426, Z    +0.000, E1   +34.947, E3 -408966.788}
SPL {X  -158.886, Y  +690.264, Z    +0.000, E1   +34.888, E3 -408978.805}
SPL {X  -158.362, Y  +694.266, Z    +0.000, E1   +34.794, E3 -408991.478}
SPL {X  -157.614, Y  +698.973, Z    +0.000, E1   +34.690, E3 -409006.479}
SPL {X  -156.901, Y  +702.787, Z    +0.000, E1   +34.523, E3 -409018.822}
SPL {X  -156.097, Y  +706.580, Z    +0.000, E1   +34.427, E3 -409031.062}
SPL {X  -155.080, Y  +710.833, Z    +0.000, E1   +34.231, E3 -409044.996}
SPL {X  -153.755, Y  +715.731, Z    +0.000, E1   +30.246, E3 -409094.262}
ENDSPLINE

SPLINE
SPL {X  -155.537, Y  +708.983, Z    +0.000, E1   +25.008, E3 -409120.089}
SPL {X  -158.838, Y  +690.666, Z    +0.000, E1   +14.584, E3 -409144.801}
SPL {X  -159.750, Y  +680.262, Z    +0.000, E1    +8.563, E3 -409150.942}
SPL {X  -159.973, Y  +673.798, Z    +0.000, E1    +4.600, E3 -409153.406}
SPL {X  -159.990, Y  +668.863, Z    +0.000, E1    +1.298, E3 -409154.845}
SPL {X  -159.990, Y  +663.839, Z    +0.000, E1    -2.454, E3 -409156.106}
SPL {X  -159.990, Y  +658.349, Z    +0.000, E1    -7.223, E3 -409157.788}
SPL {X  -159.990, Y  +650.390, Z    +0.000, E1   -14.372, E3 -409161.534}
SPL {X  -159.990, Y  +643.417, Z    +0.000, E1   -20.300, E3 -409165.798}
SPL {X  -159.990, Y  +621.124, Z    +0.000, E1   -32.598, E3 -409187.512}
SPL {X  -159.990, Y  +597.855, Z    +0.000, E1   -36.862, E3 -409230.431}
SPL {X  -159.990, Y  +592.884, Z    +0.000, E1   -36.865, E3 -409244.502}
SPL {X  -159.990, Y  +587.104, Z    +0.000, E1   -36.878, E3 -409260.859}
SPL {X  -159.990, Y  +581.795, Z    +0.000, E1   -36.847, E3 -409275.958}
SPL {X  -159.990, Y  +576.165, Z    +0.000, E1   -36.887, E3 -409291.837}
SPL {X  -159.990, Y  +570.328, Z    +0.000, E1   -36.855, E3 -409308.411}
SPL {X  -159.990, Y  +566.126, Z    +0.000, E1   -36.841, E3 -409320.317}
SPL {X  -159.990, Y  +562.387, Z    +0.000, E1   -36.853, E3 -409330.850}
SPL {X  -159.990, Y  +557.944, Z    +0.000, E1   -36.859, E3 -409343.443}
SPL {X  -159.990, Y  +552.571, Z    +0.000, E1   -36.873, E3 -409358.647}
SPL {X  -159.990, Y  +546.127, Z    +0.000, E1   -36.890, E3 -409376.874}
SPL {X  -159.990, Y  +539.889, Z    +0.000, E1   -36.872, E3 -409394.572}
SPL {X  -159.990, Y  +534.469, Z    +0.000, E1   -36.855, E3 -409409.970}
SPL {X  -159.990, Y  +528.569, Z    +0.000, E1   -36.871, E3 -409426.688}
SPL {X  -159.990, Y  +522.641, Z    +0.000, E1   -36.854, E3 -409443.499}
SPL {X  -159.990, Y  +517.225, Z    +0.000, E1   -36.859, E3 -409458.833}
SPL {X  -159.990, Y  +511.408, Z    +0.000, E1   -36.858, E3 -409475.321}
SPL {X  -159.990, Y  +505.756, Z    +0.000, E1   -36.857, E3 -409491.331}
SPL {X  -159.990, Y  +499.829, Z    +0.000, E1   -36.864, E3 -409508.136}
SPL {X  -159.990, Y  +498.054, Z    +0.000, E1   -35.692, E3 -409520.175}
ENDSPLINE

SPLINE
SPL {X  -159.990, Y  +506.994, Z    +0.000, E1   -30.162, E3 -409526.837}
ENDSPLINE

SPLINE
SPL {X  -159.990, Y  +502.084, Z    +0.000, E1   -31.057, E3 -409538.488}
SPL {X  -159.990, Y  +494.586, Z    +0.000, E1   -32.444, E3 -409555.092}
SPL {X  -159.990, Y  +486.073, Z    +0.000, E1   -33.960, E3 -409572.929}
SPL {X  -159.990, Y  +477.314, Z    +0.000, E1   -35.342, E3 -409591.108}
SPL {X  -159.990, Y  +471.459, Z    +0.000, E1   -35.779, E3 -409605.647}
SPL {X  -159.990, Y  +466.474, Z    +0.000, E1   -35.796, E3 -409620.306}
SPL {X  -159.990, Y  +461.990, Z    +0.000, E1   -35.776, E3 -409633.541}
SPL {X  -159.990, Y  +458.524, Z    +0.000, E1   -35.761, E3 -409643.778}
SPL {X  -159.990, Y  +453.597, Z    +0.000, E1   -35.819, E3 -409658.198}
SPL {X  -159.990, Y  +448.227, Z    +0.000, E1   -35.776, E3 -409674.076}
SPL {X  -159.990, Y  +443.707, Z    +0.000, E1   -35.784, E3 -409687.372}
SPL {X  -159.990, Y  +439.109, Z    +0.000, E1   -35.781, E3 -409700.908}
SPL {X  -159.990, Y  +435.535, Z    +0.000, E1   -35.764, E3 -409711.458}
SPL {X  -159.990, Y  +431.100, Z    +0.000, E1   -35.807, E3 -409724.443}
SPL {X  -159.990, Y  +425.407, Z    +0.000, E1   -35.800, E3 -409741.219}
SPL {X  -159.990, Y  +420.199, Z    +0.000, E1   -35.790, E3 -409756.573}
SPL {X  -159.990, Y  +414.514, Z    +0.000, E1   -35.815, E3 -409773.272}
SPL {X  -159.990, Y  +408.600, Z    +0.000, E1   -35.802, E3 -409790.711}
SPL {X  -159.990, Y  +403.496, Z    +0.000, E1   -35.787, E3 -409805.765}
SPL {X  -159.990, Y  +398.606, Z    +0.000, E1   -35.794, E3 -409820.153}
SPL {X  -159.990, Y  +394.138, Z    +0.000, E1   -35.778, E3 -409833.336}
SPL {X  -159.990, Y  +390.065, Z    +0.000, E1   -35.780, E3 -409845.326}
SPL {X  -159.990, Y  +385.506, Z    +0.000, E1   -35.789, E3 -409858.732}
SPL {X  -159.976, Y  +380.359, Z    +0.000, E1   -35.797, E3 -409873.881}
SPL {X  -159.831, Y  +375.358, Z    +0.000, E1   -35.763, E3 -409888.771}
SPL {X  -159.547, Y  +370.604, Z    +0.000, E1   -35.724, E3 -409903.070}
SPL {X  -159.134, Y  +365.969, Z    +0.000, E1   -35.644, E3 -409917.156}
SPL {X  -158.606, Y  +361.498, Z    +0.000, E1   -35.550, E3 -409930.920}
SPL {X  -157.918, Y  +356.833, Z    +0.000, E1   -35.439, E3 -409945.373}
SPL {X  -157.185, Y  +352.671, Z    +0.000, E1   -35.292, E3 -409958.434}
SPL {X  -156.302, Y  +348.345, Z    +0.000, E1   -35.165, E3 -409972.055}
SPL {X  -155.054, Y  +343.066, Z    +0.000, E1   -34.964, E3 -409988.870}
SPL {X  -154.305, Y  +340.232, Z    +0.000, E1   -28.975, E3 -410046.429}
ENDSPLINE

SPLINE
SPL {X  -158.456, Y  +360.399, Z    +0.000, E1   -16.490, E3 -410083.249}
SPL {X  -159.553, Y  +370.677, Z    +0.000, E1   -10.576, E3 -410091.009}
SPL {X  -159.960, Y  +379.402, Z    +0.000, E1    -5.303, E3 -410095.029}
SPL {X  -159.990, Y  +385.983, Z    +0.000, E1    -0.882, E3 -410097.102}
SPL {X  -159.990, Y  +390.933, Z    +0.000, E1    +2.877, E3 -410098.550}
SPL {X  -159.990, Y  +396.375, Z    +0.000, E1    +7.538, E3 -410100.324}
SPL {X  -159.990, Y  +405.219, Z    +0.000, E1   +15.296, E3 -410104.642}
SPL {X  -159.990, Y  +427.416, Z    +0.000, E1   +29.294, E3 -410125.697}
SPL {X  -159.990, Y  +447.483, Z    +0.000, E1   +34.518, E3 -410159.862}
SPL {X  -159.990, Y  +453.425, Z    +0.000, E1   +35.055, E3 -410174.545}
SPL {X  -159.990, Y  +457.209, Z    +0.000, E1   +35.039, E3 -410186.020}
SPL {X  -159.990, Y  +460.708, Z    +0.000, E1   +35.045, E3 -410196.602}
SPL {X  -159.990, Y  +464.162, Z    +0.000, E1   +35.038, E3 -410207.059}
SPL {X  -159.990, Y  +467.857, Z    +0.000, E1   +35.053, E3 -410218.216}
SPL {X  -159.990, Y  +471.326, Z    +0.000, E1   +35.038, E3 -410228.711}
SPL {X  -159.990, Y  +474.610, Z    +0.000, E1   +35.053, E3 -410238.610}
SPL {X  -159.990, Y  +478.303, Z    +0.000, E1   +35.049, E3 -410249.782}
SPL {X  -159.990, Y  +482.537, Z    +0.000, E1   +35.066, E3 -410262.574}
SPL {X  -159.990, Y  +487.181, Z    +0.000, E1   +35.054, E3 -410276.657}
SPL {X  -159.990, Y  +492.368, Z    +0.000, E1   +35.076, E3 -410292.329}
SPL {X  -159.990, Y  +497.072, Z    +0.000, E1   +35.040, E3 -410306.625}
SPL {X  -159.990, Y  +501.645, Z    +0.000, E1   +35.067, E3 -410320.408}
SPL {X  -159.990, Y  +506.307, Z    +0.000, E1   +35.049, E3 -410334.530}
SPL {X  -159.990, Y  +511.643, Z    +0.000, E1   +35.091, E3 -410350.610}
SPL {X  -159.990, Y  +517.156, Z    +0.000, E1   +35.059, E3 -410367.328}
SPL {X  -159.990, Y  +521.637, Z    +0.000, E1   +35.056, E3 -410380.891}
SPL {X  -159.990, Y  +526.246, Z    +0.000, E1   +35.065, E3 -410394.795}
SPL {X  -159.990, Y  +530.289, Z    +0.000, E1   +35.044, E3 -410407.081}
SPL {X  -159.990, Y  +534.797, Z    +0.000, E1   +35.069, E3 -410420.681}
SPL {X  -159.990, Y  +538.710, Z    +0.000, E1   +35.033, E3 -410432.578}
SPL {X  -159.990, Y  +542.114, Z    +0.000, E1   +35.053, E3 -410442.830}
SPL {X  -159.990, Y  +546.612, Z    +0.000, E1   +35.065, E3 -410456.402}
SPL {X  -159.990, Y  +551.596, Z    +0.000, E1   +35.079, E3 -410471.437}
SPL {X  -159.990, Y  +556.051, Z    +0.000, E1   +35.060, E3 -410484.899}
SPL {X  -159.990, Y  +560.931, Z    +0.000, E1   +35.098, E3 -410499.604}
SPL {X  -159.990, Y  +564.815, Z    +0.000, E1   +35.041, E3 -410511.452}
SPL {X  -159.990, Y  +567.494, Z    +0.000, E1   +35.052, E3 -410519.533}
SPL {X  -159.990, Y  +571.374, Z    +0.000, E1   +35.070, E3 -410531.236}
SPL {X  -159.990, Y  +575.771, Z    +0.000, E1   +35.064, E3 -410544.541}
SPL {X  -159.990, Y  +580.750, Z    +0.000, E1   +35.087, E3 -410559.563}
SPL {X  -159.990, Y  +585.414, Z    +0.000, E1   +35.059, E3 -410573.709}
SPL {X  -159.990, Y  +590.166, Z    +0.000, E1   +35.084, E3 -410588.038}
SPL {X  -159.990, Y  +595.313, Z    +0.000, E1   +35.073, E3 -410603.617}
SPL {X  -159.990, Y  +599.479, Z    +0.000, E1   +35.059, E3 -410616.234}
SPL {X  -159.990, Y  +603.289, Z    +0.000, E1   +35.068, E3 -410627.723}
SPL {X  -159.990, Y  +607.919, Z    +0.000, E1   +35.079, E3 -410641.712}
SPL {X  -159.990, Y  +613.036, Z    +0.000, E1   +35.082, E3 -410657.183}
SPL {X  -159.990, Y  +617.577, Z    +0.000, E1   +35.061, E3 -410670.944}
SPL {X  -159.990, Y  +621.534, Z    +0.000, E1   +35.068, E3 -410682.878}
SPL {X  -159.990, Y  +626.426, Z    +0.000, E1   +35.093, E3 -410697.638}
SPL {X  -159.990, Y  +631.553, Z    +0.000, E1   +35.068, E3 -410713.196}
SPL {X  -159.990, Y  +635.965, Z    +0.000, E1   +35.065, E3 -410726.544}
SPL {X  -159.990, Y  +640.633, Z    +0.000, E1   +35.080, E3 -410740.632}
SPL {X  -159.990, Y  +645.423, Z    +0.000, E1   +35.070, E3 -410755.138}
SPL {X  -159.990, Y  +650.555, Z    +0.000, E1   +35.089, E3 -410770.627}
SPL {X  -159.990, Y  +656.270, Z    +0.000, E1   +35.087, E3 -410787.920}
SPL {X  -159.990, Y  +661.105, Z    +0.000, E1   +35.059, E3 -410802.584}
SPL {X  -159.990, Y  +665.311, Z    +0.000, E1   +35.064, E3 -410815.298}
SPL {X  -159.990, Y  +670.193, Z    +0.000, E1   +35.076, E3 -410830.046}
SPL {X  -159.948, Y  +675.148, Z    +0.000, E1   +35.069, E3 -410845.038}
SPL {X  -159.752, Y  +680.228, Z    +0.000, E1   +35.050, E3 -410860.585}
SPL {X  -159.371, Y  +685.563, Z    +0.000, E1   +34.989, E3 -410877.097}
SPL {X  -158.886, Y  +690.264, Z    +0.000, E1   +34.888, E3 -410891.848}
SPL {X  -158.362, Y  +694.266, Z    +0.000, E1   +34.794, E3 -410904.522}
SPL {X  -157.614, Y  +698.973, Z    +0.000, E1   +34.690, E3 -410919.522}
SPL {X  -156.640, Y  +704.066, Z    +0.000, E1   +34.516, E3 -410935.947}
SPL {X  -155.835, Y  +707.723, Z    +0.000, E1   +34.344, E3 -410947.890}
SPL {X  -155.153, Y  +710.542, Z    +0.000, E1   +34.234, E3 -410957.109}
SPL {X  -153.767, Y  +715.686, Z    +0.000, E1   +30.747, E3 -411002.327}
ENDSPLINE

SPLINE
SPL {X  -154.589, Y  +712.719, Z    +0.000, E1   +27.400, E3 -411023.728}
SPL {X  -158.529, Y  +693.075, Z    +0.000, E1   +15.996, E3 -411055.574}
SPL {X  -159.750, Y  +680.262, Z    +0.000, E1    +8.563, E3 -411063.985}
SPL {X  -159.973, Y  +673.798, Z    +0.000, E1    +4.600, E3 -411066.449}
SPL {X  -159.990, Y  +667.448, Z    +0.000, E1    +0.356, E3 -411068.229}
SPL {X  -159.990, Y  +662.686, Z    +0.000, E1    -3.472, E3 -411069.464}
SPL {X  -159.990, Y  +658.349, Z    +0.000, E1    -7.223, E3 -411070.832}
SPL {X  -159.990, Y  +653.910, Z    +0.000, E1   -11.344, E3 -411072.600}
SPL {X  -159.990, Y  +646.193, Z    +0.000, E1   -17.980, E3 -411077.069}
SPL {X  -159.990, Y  +621.124, Z    +0.000, E1   -32.598, E3 -411100.556}
SPL {X  -159.990, Y  +597.855, Z    +0.000, E1   -36.862, E3 -411143.475}
SPL {X  -159.990, Y  +592.884, Z    +0.000, E1   -36.865, E3 -411157.546}
SPL {X  -159.990, Y  +587.104, Z    +0.000, E1   -36.878, E3 -411173.903}
SPL {X  -159.990, Y  +581.795, Z    +0.000, E1   -36.847, E3 -411189.001}
SPL {X  -159.990, Y  +576.165, Z    +0.000, E1   -36.887, E3 -411204.881}
SPL {X  -159.990, Y  +570.328, Z    +0.000, E1   -36.855, E3 -411221.454}
SPL {X  -159.990, Y  +566.126, Z    +0.000, E1   -36.841, E3 -411233.360}
SPL {X  -159.990, Y  +562.387, Z    +0.000, E1   -36.853, E3 -411243.893}
SPL {X  -159.990, Y  +557.944, Z    +0.000, E1   -36.859, E3 -411256.487}
SPL {X  -159.990, Y  +553.661, Z    +0.000, E1   -36.844, E3 -411268.650}
SPL {X  -159.990, Y  +549.195, Z    +0.000, E1   -36.856, E3 -411281.286}
SPL {X  -159.990, Y  +543.458, Z    +0.000, E1   -36.882, E3 -411297.484}
SPL {X  -159.990, Y  +537.639, Z    +0.000, E1   -36.860, E3 -411314.022}
SPL {X  -159.990, Y  +531.894, Z    +0.000, E1   -36.865, E3 -411330.311}
SPL {X  -159.990, Y  +527.151, Z    +0.000, E1   -36.828, E3 -411343.810}
SPL {X  -159.990, Y  +522.641, Z    +0.000, E1   -36.854, E3 -411356.542}
SPL {X  -159.990, Y  +517.225, Z    +0.000, E1   -36.859, E3 -411371.877}
SPL {X  -159.990, Y  +512.789, Z    +0.000, E1   -36.824, E3 -411384.504}
SPL {X  -159.990, Y  +508.591, Z    +0.000, E1   -36.846, E3 -411396.367}
SPL {X  -159.990, Y  +503.454, Z    +0.000, E1   -36.847, E3 -411410.922}
SPL {X  -159.990, Y  +498.817, Z    +0.000, E1   -36.830, E3 -411424.105}
SPL {X  -159.990, Y  +498.054, Z    +0.000, E1   -35.692, E3 -411433.219}
ENDSPLINE

SPLINE
SPL {X  -159.990, Y  +506.994, Z    +0.000, E1   -30.162, E3 -411439.880}
ENDSPLINE

SPLINE
SPL {X  -159.990, Y  +502.084, Z    +0.000, E1   -31.057, E3 -411451.532}
SPL {X  -159.990, Y  +494.586, Z    +0.000, E1   -32.444, E3 -411468.135}
SPL {X  -159.990, Y  +487.723, Z    +0.000, E1   -33.658, E3 -411482.588}
SPL {X  -159.990, Y  +481.374, Z    +0.000, E1   -34.706, E3 -411495.792}
SPL {X  -159.990, Y  +475.503, Z    +0.000, E1   -35.597, E3 -411507.844}
SPL {X  -159.990, Y  +471.459, Z    +0.000, E1   -35.779, E3 -411518.691}
SPL {X  -159.990, Y  +467.485, Z    +0.000, E1   -35.768, E3 -411530.420}
SPL {X  -159.990, Y  +462.739, Z    +0.000, E1   -35.799, E3 -411544.348}
SPL {X  -159.990, Y  +457.385, Z    +0.000, E1   -35.788, E3 -411560.132}
SPL {X  -159.990, Y  +452.637, Z    +0.000, E1   -35.783, E3 -411574.123}
SPL {X  -159.990, Y  +448.227, Z    +0.000, E1   -35.776, E3 -411587.120}
SPL {X  -159.990, Y  +443.707, Z    +0.000, E1   -35.784, E3 -411600.415}
SPL {X  -159.990, Y  +439.109, Z    +0.000, E1   -35.781, E3 -411613.951}
SPL {X  -159.990, Y  +434.400, Z    +0.000, E1   -35.789, E3 -411627.806}
SPL {X  -159.990, Y  +430.115, Z    +0.000, E1   -35.777, E3 -411640.423}
SPL {X  -159.990, Y  +426.641, Z    +0.000, E1   -35.769, E3 -411650.674}
SPL {X  -159.990, Y  +422.627, Z    +0.000, E1   -35.788, E3 -411662.471}
SPL {X  -159.990, Y  +417.866, Z    +0.000, E1   -35.788, E3 -411676.484}
SPL {X  -159.990, Y  +413.498, Z    +0.000, E1   -35.779, E3 -411689.366}
SPL {X  -159.990, Y  +408.600, Z    +0.000, E1   -35.802, E3 -411703.754}
SPL {X  -159.990, Y  +403.496, Z    +0.000, E1   -35.787, E3 -411718.809}
SPL {X  -159.990, Y  +398.606, Z    +0.000, E1   -35.794, E3 -411733.196}
SPL {X  -159.990, Y  +394.138, Z    +0.000, E1   -35.778, E3 -411746.379}
SPL {X  -159.990, Y  +390.065, Z    +0.000, E1   -35.780, E3 -411758.370}
SPL {X  -159.990, Y  +385.506, Z    +0.000, E1   -35.789, E3 -411771.775}
SPL {X  -159.989, Y  +381.970, Z    +0.000, E1   -35.761, E3 -411782.230}
SPL {X  -159.936, Y  +378.352, Z    +0.000, E1   -35.782, E3 -411792.885}
SPL {X  -159.790, Y  +374.497, Z    +0.000, E1   -35.735, E3 -411804.429}
SPL {X  -159.547, Y  +370.604, Z    +0.000, E1   -35.724, E3 -411816.114}
SPL {X  -159.134, Y  +365.969, Z    +0.000, E1   -35.644, E3 -411830.199}
SPL {X  -158.606, Y  +361.498, Z    +0.000, E1   -35.550, E3 -411843.964}
SPL {X  -157.918, Y  +356.833, Z    +0.000, E1   -35.439, E3 -411858.417}
SPL {X  -157.185, Y  +352.671, Z    +0.000, E1   -35.292, E3 -411871.477}
SPL {X  -156.302, Y  +348.345, Z    +0.000, E1   -35.165, E3 -411885.098}
SPL {X  -155.054, Y  +343.066, Z    +0.000, E1   -34.964, E3 -411901.913}
SPL {X  -154.305, Y  +340.232, Z    +0.000, E1   -28.975, E3 -411959.473}
ENDSPLINE

SPLINE
SPL {X  -158.456, Y  +360.399, Z    +0.000, E1   -16.490, E3 -411996.293}
SPL {X  -159.553, Y  +370.677, Z    +0.000, E1   -10.576, E3 -412004.053}
SPL {X  -159.960, Y  +379.402, Z    +0.000, E1    -5.303, E3 -412008.073}
SPL {X  -159.990, Y  +387.301, Z    +0.000, E1    -0.001, E3 -412010.534}
SPL {X  -159.990, Y  +392.161, Z    +0.000, E1    +3.946, E3 -412011.946}
SPL {X  -159.990, Y  +396.375, Z    +0.000, E1    +7.538, E3 -412013.368}
SPL {X  -159.990, Y  +404.277, Z    +0.000, E1   +14.543, E3 -412017.031}
SPL {X  -159.990, Y  +423.101, Z    +0.000, E1   +27.351, E3 -412033.470}
SPL {X  -159.990, Y  +430.933, Z    +0.000, E1   +30.672, E3 -412043.441}
SPL {X  -159.990, Y  +451.842, Z    +0.000, E1   +35.050, E3 -412082.812}
SPL {X  -159.990, Y  +456.402, Z    +0.000, E1   +35.061, E3 -412096.588}
SPL {X  -159.990, Y  +460.708, Z    +0.000, E1   +35.045, E3 -412109.646}
SPL {X  -159.990, Y  +465.240, Z    +0.000, E1   +35.066, E3 -412123.321}
SPL {X  -159.990, Y  +470.278, Z    +0.000, E1   +35.063, E3 -412138.555}
SPL {X  -159.990, Y  +474.610, Z    +0.000, E1   +35.053, E3 -412151.654}
SPL {X  -159.990, Y  +478.303, Z    +0.000, E1   +35.049, E3 -412162.826}
SPL {X  -159.990, Y  +482.537, Z    +0.000, E1   +35.066, E3 -412175.617}
SPL {X  -159.990, Y  +487.181, Z    +0.000, E1   +35.054, E3 -412189.700}
SPL {X  -159.990, Y  +490.807, Z    +0.000, E1   +35.036, E3 -412200.701}
SPL {X  -159.990, Y  +493.669, Z    +0.000, E1   +35.034, E3 -412209.381}
SPL {X  -159.990, Y  +497.072, Z    +0.000, E1   +35.040, E3 -412219.668}
SPL {X  -159.990, Y  +500.395, Z    +0.000, E1   +35.033, E3 -412229.731}
SPL {X  -159.990, Y  +502.996, Z    +0.000, E1   +35.034, E3 -412237.579}
SPL {X  -159.990, Y  +507.359, Z    +0.000, E1   +35.080, E3 -412250.708}
SPL {X  -159.990, Y  +512.562, Z    +0.000, E1   +35.055, E3 -412266.490}
SPL {X  -159.990, Y  +517.156, Z    +0.000, E1   +35.059, E3 -412280.371}
SPL {X  -159.990, Y  +521.637, Z    +0.000, E1   +35.056, E3 -412293.935}
SPL {X  -159.990, Y  +525.227, Z    +0.000, E1   +35.041, E3 -412304.795}
SPL {X  -159.990, Y  +529.413, Z    +0.000, E1   +35.072, E3 -412317.424}
SPL {X  -159.990, Y  +534.797, Z    +0.000, E1   +35.069, E3 -412333.725}
SPL {X  -159.990, Y  +538.710, Z    +0.000, E1   +35.033, E3 -412345.622}
SPL {X  -159.990, Y  +542.114, Z    +0.000, E1   +35.053, E3 -412355.874}
SPL {X  -159.990, Y  +545.724, Z    +0.000, E1   +35.043, E3 -412366.798}
SPL {X  -159.990, Y  +549.546, Z    +0.000, E1   +35.061, E3 -412378.323}
SPL {X  -159.990, Y  +554.793, Z    +0.000, E1   +35.100, E3 -412394.086}
SPL {X  -159.990, Y  +560.931, Z    +0.000, E1   +35.098, E3 -412412.648}
SPL {X  -159.990, Y  +566.542, Z    +0.000, E1   +35.080, E3 -412429.655}
SPL {X  -159.990, Y  +570.261, Z    +0.000, E1   +35.046, E3 -412440.951}
SPL {X  -159.990, Y  +574.780, Z    +0.000, E1   +35.101, E3 -412454.531}
SPL {X  -159.990, Y  +580.750, Z    +0.000, E1   +35.087, E3 -412472.607}
SPL {X  -159.990, Y  +585.414, Z    +0.000, E1   +35.059, E3 -412486.753}
SPL {X  -159.990, Y  +588.716, Z    +0.000, E1   +35.047, E3 -412496.756}
SPL {X  -159.990, Y  +591.475, Z    +0.000, E1   +35.047, E3 -412505.096}
SPL {X  -159.990, Y  +595.313, Z    +0.000, E1   +35.073, E3 -412516.660}
SPL {X  -159.990, Y  +600.543, Z    +0.000, E1   +35.091, E3 -412532.443}
SPL {X  -159.990, Y  +605.846, Z    +0.000, E1   +35.077, E3 -412548.494}
SPL {X  -159.990, Y  +609.372, Z    +0.000, E1   +35.047, E3 -412559.192}
SPL {X  -159.990, Y  +613.036, Z    +0.000, E1   +35.082, E3 -412570.226}
SPL {X  -159.990, Y  +617.577, Z    +0.000, E1   +35.061, E3 -412583.988}
SPL {X  -159.990, Y  +621.534, Z    +0.000, E1   +35.068, E3 -412595.922}
SPL {X  -159.990, Y  +625.237, Z    +0.000, E1   +35.062, E3 -412607.124}
SPL {X  -159.990, Y  +629.217, Z    +0.000, E1   +35.065, E3 -412619.181}
SPL {X  -159.990, Y  +632.566, Z    +0.000, E1   +35.044, E3 -412629.344}
SPL {X  -159.990, Y  +635.965, Z    +0.000, E1   +35.065, E3 -412639.588}
SPL {X  -159.990, Y  +640.633, Z    +0.000, E1   +35.080, E3 -412653.676}
SPL {X  -159.990, Y  +646.430, Z    +0.000, E1   +35.102, E3 -412671.177}
SPL {X  -159.990, Y  +651.502, Z    +0.000, E1   +35.058, E3 -412686.587}
SPL {X  -159.990, Y  +654.793, Z    +0.000, E1   +35.049, E3 -412696.550}
SPL {X  -159.990, Y  +657.535, Z    +0.000, E1   +35.049, E3 -412704.847}
SPL {X  -159.990, Y  +661.105, Z    +0.000, E1   +35.059, E3 -412715.627}
SPL {X  -159.990, Y  +665.311, Z    +0.000, E1   +35.064, E3 -412728.342}
SPL {X  -159.990, Y  +668.650, Z    +0.000, E1   +35.040, E3 -412738.482}
SPL {X  -159.990, Y  +671.288, Z    +0.000, E1   +35.046, E3 -412746.446}
SPL {X  -159.948, Y  +675.148, Z    +0.000, E1   +35.069, E3 -412758.081}
SPL {X  -159.752, Y  +680.228, Z    +0.000, E1   +35.050, E3 -412773.629}
SPL {X  -159.371, Y  +685.563, Z    +0.000, E1   +34.989, E3 -412790.140}
SPL {X  -158.886, Y  +690.264, Z    +0.000, E1   +34.888, E3 -412804.892}
SPL {X  -158.362, Y  +694.266, Z    +0.000, E1   +34.794, E3 -412817.565}
SPL {X  -157.614, Y  +698.973, Z    +0.000, E1   +34.690, E3 -412832.566}
SPL {X  -156.640, Y  +704.066, Z    +0.000, E1   +34.516, E3 -412848.991}
SPL {X  -155.835, Y  +707.723, Z    +0.000, E1   +34.344, E3 -412860.933}
SPL {X  -155.080, Y  +710.833, Z    +0.000, E1   +34.231, E3 -412871.083}
SPL {X  -153.949, Y  +715.047, Z    +0.000, E1   +29.578, E3 -412924.633}
ENDSPLINE

SPLINE
SPL {X  -158.529, Y  +693.075, Z    +0.000, E1   +15.996, E3 -412968.618}
SPL {X  -159.750, Y  +680.262, Z    +0.000, E1    +8.563, E3 -412977.029}
SPL {X  -159.973, Y  +673.798, Z    +0.000, E1    +4.600, E3 -412979.493}
SPL {X  -159.990, Y  +668.863, Z    +0.000, E1    +1.298, E3 -412980.932}
SPL {X  -159.990, Y  +663.839, Z    +0.000, E1    -2.454, E3 -412982.193}
SPL {X  -159.990, Y  +658.349, Z    +0.000, E1    -7.223, E3 -412983.875}
SPL {X  -159.990, Y  +650.390, Z    +0.000, E1   -14.372, E3 -412987.621}
SPL {X  -159.990, Y  +643.417, Z    +0.000, E1   -20.300, E3 -412991.885}
SPL {X  -159.990, Y  +621.124, Z    +0.000, E1   -32.598, E3 -413013.599}
SPL {X  -159.990, Y  +597.855, Z    +0.000, E1   -36.862, E3 -413056.518}
SPL {X  -159.990, Y  +593.971, Z    +0.000, E1   -36.841, E3 -413067.551}
SPL {X  -159.990, Y  +589.749, Z    +0.000, E1   -36.860, E3 -413079.478}
SPL {X  -159.990, Y  +585.754, Z    +0.000, E1   -36.838, E3 -413090.833}
SPL {X  -159.990, Y  +581.795, Z    +0.000, E1   -36.847, E3 -413102.045}
SPL {X  -159.990, Y  +577.286, Z    +0.000, E1   -36.853, E3 -413114.802}
SPL {X  -159.990, Y  +572.409, Z    +0.000, E1   -36.854, E3 -413128.614}
SPL {X  -159.990, Y  +567.110, Z    +0.000, E1   -36.868, E3 -413143.575}
SPL {X  -159.990, Y  +562.387, Z    +0.000, E1   -36.853, E3 -413156.937}
SPL {X  -159.990, Y  +557.944, Z    +0.000, E1   -36.859, E3 -413169.530}
SPL {X  -159.990, Y  +553.661, Z    +0.000, E1   -36.844, E3 -413181.694}
SPL {X  -159.990, Y  +549.195, Z    +0.000, E1   -36.856, E3 -413194.329}
SPL {X  -159.990, Y  +544.733, Z    +0.000, E1   -36.845, E3 -413206.975}
SPL {X  -159.990, Y  +539.889, Z    +0.000, E1   -36.872, E3 -413220.659}
SPL {X  -159.990, Y  +534.469, Z    +0.000, E1   -36.855, E3 -413236.057}
SPL {X  -159.990, Y  +530.428, Z    +0.000, E1   -36.821, E3 -413247.591}
SPL {X  -159.990, Y  +525.940, Z    +0.000, E1   -36.859, E3 -413260.237}
SPL {X  -159.990, Y  +520.301, Z    +0.000, E1   -36.855, E3 -413276.213}
SPL {X  -159.990, Y  +516.005, Z    +0.000, E1   -36.824, E3 -413288.440}
SPL {X  -159.990, Y  +511.408, Z    +0.000, E1   -36.858, E3 -413301.408}
SPL {X  -159.990, Y  +505.756, Z    +0.000, E1   -36.857, E3 -413317.418}
SPL {X  -159.990, Y  +499.829, Z    +0.000, E1   -36.864, E3 -413334.223}
SPL {X  -159.990, Y  +498.054, Z    +0.000, E1   -35.692, E3 -413346.262}
ENDSPLINE

SPLINE
SPL {X  -159.990, Y  +505.140, Z    +0.000, E1   -30.523, E3 -413357.289}
ENDSPLINE

